LIN {X 0,Y 456.194,Z 627.483,A -85,B 0,C 180,E1 -8384.954,E2 -8384.954} C_VEL
LIN {X 0,Y 456.575,Z 617.149,A -85,B 0,C 180,E1 -8385.37,E2 -8385.37} C_VEL
LIN {X 0,Y 456.808,Z 606.428,A -85,B 0,C 180,E1 -8385.676,E2 -8385.676} C_VEL
LIN {X 0,Y 457.125,Z 587.235,A -85,B 0,C 180,E1 -8386.008,E2 -8386.008} C_VEL
LIN {X 0,Y 457.499,Z 519.528,A -85,B 0,C 180,E1 -8387.08,E2 -8387.08} C_VEL
LIN {X 0,Y 453.991,Z 499.289,A -85,B 0,C 180,E1 -8387.558,E2 -8387.558} C_VEL
LIN {X 0,Y 453.961,Z 498.233,A -85,B 0,C 180,E1 -8387.695,E2 -8387.695} C_VEL
LIN {X 0,Y 454.542,Z 486.824,A -85,B 0,C 180,E1 -8390.358,E2 -8390.358} C_VEL
LIN {X 0,Y 455.179,Z 474.408,A -85,B 0,C 180,E1 -8393.186,E2 -8393.186} C_VEL
LIN {X 0,Y 455.543,Z 466.02,A -85,B 0,C 180,E1 -8395.104,E2 -8395.104} C_VEL
LIN {X 0,Y 453.728,Z 455.779,A -85,B 0,C 180,E1 -8397.689,E2 -8397.689} C_VEL
LIN {X 0,Y 453.526,Z 454.578,A -85,B 0,C 180,E1 -8398.078,E2 -8398.078} C_VEL
LIN {X 0,Y 453.466,Z 454.501,A -85,B 0,C 180,E1 -8401.524,E2 -8401.524} C_VEL
LIN {X 0,Y 453.481,Z 454.495,A -85,B 0,C 180,E1 -8404.775,E2 -8404.775} C_VEL
LIN {X 0,Y 453.442,Z 454.504,A -85,B 0,C 180,E1 -8408.313,E2 -8408.313} C_VEL
LIN {X 0,Y 453.465,Z 454.484,A -85,B 0,C 180,E1 -8410.612,E2 -8410.612} C_VEL
LIN {X 0,Y 453.476,Z 454.496,A -85,B 0,C 180,E1 -8414.527,E2 -8414.527} C_VEL
LIN {X 0,Y 453.431,Z 454.507,A -85,B 0,C 180,E1 -8418.071,E2 -8418.071} C_VEL
LIN {X 0,Y 453.423,Z 454.498,A -85,B 0,C 180,E1 -8420.804,E2 -8420.804} C_VEL
LIN {X 0,Y 453.44,Z 454.505,A -85,B 0,C 180,E1 -8423.915,E2 -8423.915} C_VEL
LIN {X 0,Y 453.472,Z 454.489,A -85,B 0,C 180,E1 -8427.149,E2 -8427.149} C_VEL
LIN {X 0,Y 453.46,Z 454.5,A -85,B 0,C 180,E1 -8430.266,E2 -8430.266} C_VEL
LIN {X 0,Y 453.437,Z 454.486,A -85,B 0,C 180,E1 -8433.288,E2 -8433.288} C_VEL
LIN {X 0,Y 453.491,Z 454.497,A -85,B 0,C 180,E1 -8436.237,E2 -8436.237} C_VEL
LIN {X 0,Y 453.433,Z 454.495,A -85,B 0,C 180,E1 -8439.114,E2 -8439.114} C_VEL
LIN {X 0,Y 453.452,Z 454.485,A -85,B 0,C 180,E1 -8441.941,E2 -8441.941} C_VEL
LIN {X 0,Y 453.483,Z 454.492,A -85,B 0,C 180,E1 -8444.723,E2 -8444.723} C_VEL
LIN {X 0,Y 453.562,Z 454.482,A -85,B 0,C 180,E1 -8447.47,E2 -8447.47} C_VEL
LIN {X 0,Y 453.551,Z 454.467,A -85,B 0,C 180,E1 -8451.085,E2 -8451.085} C_VEL
LIN {X 0,Y 453.629,Z 454.474,A -85,B 0,C 180,E1 -8453.773,E2 -8453.773} C_VEL
LIN {X 0,Y 453.696,Z 454.465,A -85,B 0,C 180,E1 -8457.335,E2 -8457.335} C_VEL
LIN {X 0,Y 453.742,Z 454.449,A -85,B 0,C 180,E1 -8459.999,E2 -8459.999} C_VEL
LIN {X 0,Y 453.695,Z 454.464,A -85,B 0,C 180,E1 -8462.662,E2 -8462.662} C_VEL
LIN {X 0,Y 453.628,Z 454.479,A -85,B 0,C 180,E1 -8466.225,E2 -8466.225} C_VEL
LIN {X 0,Y 453.547,Z 454.473,A -85,B 0,C 180,E1 -8468.913,E2 -8468.913} C_VEL
LIN {X 0,Y 453.557,Z 454.484,A -85,B 0,C 180,E1 -8472.527,E2 -8472.527} C_VEL
LIN {X 0,Y 453.488,Z 454.495,A -85,B 0,C 180,E1 -8476.196,E2 -8476.196} C_VEL
LIN {X 0,Y 453.476,Z 454.478,A -85,B 0,C 180,E1 -8479.026,E2 -8479.026} C_VEL
LIN {X 0,Y 453.464,Z 454.495,A -85,B 0,C 180,E1 -8481.835,E2 -8481.835} C_VEL
LIN {X 0,Y 453.457,Z 454.495,A -85,B 0,C 180,E1 -8484.736,E2 -8484.736} C_VEL
LIN {X 0,Y 453.45,Z 454.49,A -85,B 0,C 180,E1 -8487.941,E2 -8487.941} C_VEL
LIN {X 0,Y 453.445,Z 454.499,A -85,B 0,C 180,E1 -8490.76,E2 -8490.76} C_VEL
LIN {X 0,Y 453.452,Z 454.495,A -85,B 0,C 180,E1 -8493.913,E2 -8493.913} C_VEL
LIN {X 0,Y 453.422,Z 454.501,A -85,B 0,C 180,E1 -8497.19,E2 -8497.19} C_VEL
LIN {X 0,Y 453.456,Z 454.491,A -85,B 0,C 180,E1 -8500.611,E2 -8500.611} C_VEL
LIN {X 0,Y 453.466,Z 454.495,A -85,B 0,C 180,E1 -8504.527,E2 -8504.527} C_VEL
LIN {X 0,Y 453.415,Z 454.481,A -85,B 0,C 180,E1 -8508.071,E2 -8508.071} C_VEL
LIN {X 0,Y 453.41,Z 454.502,A -85,B 0,C 180,E1 -8510.803,E2 -8510.803} C_VEL
LIN {X 0,Y 453.425,Z 454.497,A -85,B 0,C 180,E1 -8513.915,E2 -8513.915} C_VEL
LIN {X 0,Y 453.456,Z 454.495,A -85,B 0,C 180,E1 -8517.149,E2 -8517.149} C_VEL
LIN {X 0,Y 453.444,Z 454.491,A -85,B 0,C 180,E1 -8520.266,E2 -8520.266} C_VEL
LIN {X 0,Y 453.425,Z 454.503,A -85,B 0,C 180,E1 -8523.289,E2 -8523.289} C_VEL
LIN {X 0,Y 453.476,Z 454.501,A -85,B 0,C 180,E1 -8526.238,E2 -8526.238} C_VEL
LIN {X 0,Y 453.464,Z 454.498,A -85,B 0,C 180,E1 -8529.117,E2 -8529.117} C_VEL
LIN {X 0,Y 453.469,Z 454.502,A -85,B 0,C 180,E1 -8531.943,E2 -8531.943} C_VEL
LIN {X 0,Y 453.503,Z 454.495,A -85,B 0,C 180,E1 -8534.725,E2 -8534.725} C_VEL
LIN {X 0,Y 453.527,Z 454.494,A -85,B 0,C 180,E1 -8538.378,E2 -8538.378} C_VEL
LIN {X 0,Y 453.553,Z 454.488,A -85,B 0,C 180,E1 -8541.086,E2 -8541.086} C_VEL
LIN {X 0,Y 453.568,Z 454.487,A -85,B 0,C 180,E1 -8543.052,E2 -8543.052} C_VEL
LIN {X 0,Y 452.886,Z 454.575,A -85,B 0,C 180,E1 -8543.794,E2 -8543.794} C_VEL
LIN {X 0,Y 449.936,Z 454.939,A -85,B 0,C 180,E1 -8544.996,E2 -8544.996} C_VEL
LIN {X 0,Y 447.507,Z 455.245,A -85,B 0,C 180,E1 -8545.965,E2 -8545.965} C_VEL
LIN {X 0,Y 446.564,Z 455.361,A -85,B 0,C 180,E1 -8546.716,E2 -8546.716} C_VEL
LIN {X 0,Y 446.541,Z 455.362,A -85,B 0,C 180,E1 -8546.97,E2 -8546.97} C_VEL
LIN {X 0,Y 446.701,Z 455.345,A -85,B 0,C 180,E1 -8550,E2 -8550} C_VEL
LIN {X 0,Y 446.635,Z 455.351,A -85,B 0,C 180,E1 -8552.706,E2 -8552.706} C_VEL
LIN {X 0,Y 446.589,Z 455.359,A -85,B 0,C 180,E1 -8556.324,E2 -8556.324} C_VEL
LIN {X 0,Y 446.501,Z 455.367,A -85,B 0,C 180,E1 -8559.056,E2 -8559.056} C_VEL
LIN {X 0,Y 446.505,Z 455.367,A -85,B 0,C 180,E1 -8562.73,E2 -8562.73} C_VEL
LIN {X 0,Y 446.437,Z 455.378,A -85,B 0,C 180,E1 -8566.209,E2 -8566.209} C_VEL
LIN {X 0,Y 446.452,Z 455.373,A -85,B 0,C 180,E1 -8569.304,E2 -8569.304} C_VEL
LIN {X 0,Y 446.4,Z 455.382,A -85,B 0,C 180,E1 -8572.2,E2 -8572.2} C_VEL
LIN {X 0,Y 446.405,Z 455.378,A -85,B 0,C 180,E1 -8575.155,E2 -8575.155} C_VEL
LIN {X 0,Y 446.401,Z 455.373,A -85,B 0,C 180,E1 -8578.184,E2 -8578.184} C_VEL
LIN {X 0,Y 446.391,Z 455.378,A -85,B 0,C 180,E1 -8581.302,E2 -8581.302} C_VEL
LIN {X 0,Y 446.404,Z 455.361,A -85,B 0,C 180,E1 -8584.525,E2 -8584.525} C_VEL
LIN {X 0,Y 446.38,Z 455.385,A -85,B 0,C 180,E1 -8588.077,E2 -8588.077} C_VEL
LIN {X 0,Y 446.38,Z 455.36,A -85,B 0,C 180,E1 -8591.396,E2 -8591.396} C_VEL
LIN {X 0,Y 446.407,Z 455.372,A -85,B 0,C 180,E1 -8595.109,E2 -8595.109} C_VEL
LIN {X 0,Y 446.386,Z 455.371,A -85,B 0,C 180,E1 -8598.607,E2 -8598.607} C_VEL
LIN {X 0,Y 446.384,Z 455.385,A -85,B 0,C 180,E1 -8601.925,E2 -8601.925} C_VEL
LIN {X 0,Y 446.407,Z 455.368,A -85,B 0,C 180,E1 -8605.477,E2 -8605.477} C_VEL
LIN {X 0,Y 446.395,Z 455.377,A -85,B 0,C 180,E1 -8608.7,E2 -8608.7} C_VEL
LIN {X 0,Y 446.413,Z 455.368,A -85,B 0,C 180,E1 -8611.838,E2 -8611.838} C_VEL
LIN {X 0,Y 446.409,Z 455.372,A -85,B 0,C 180,E1 -8614.847,E2 -8614.847} C_VEL
LIN {X 0,Y 446.437,Z 455.369,A -85,B 0,C 180,E1 -8618.247,E2 -8618.247} C_VEL
LIN {X 0,Y 446.4,Z 455.363,A -85,B 0,C 180,E1 -8621.648,E2 -8621.648} C_VEL
LIN {X 0,Y 446.446,Z 455.372,A -85,B 0,C 180,E1 -8624.479,E2 -8624.479} C_VEL
LIN {X 0,Y 446.509,Z 455.361,A -85,B 0,C 180,E1 -8627.386,E2 -8627.386} C_VEL
LIN {X 0,Y 446.498,Z 455.351,A -85,B 0,C 180,E1 -8630.945,E2 -8630.945} C_VEL
LIN {X 0,Y 446.598,Z 455.353,A -85,B 0,C 180,E1 -8633.677,E2 -8633.677} C_VEL
LIN {X 0,Y 446.644,Z 455.342,A -85,B 0,C 180,E1 -8637.296,E2 -8637.296} C_VEL
LIN {X 0,Y 446.693,Z 455.326,A -85,B 0,C 180,E1 -8640.001,E2 -8640.001} C_VEL
LIN {X 0,Y 446.645,Z 455.343,A -85,B 0,C 180,E1 -8642.707,E2 -8642.707} C_VEL
LIN {X 0,Y 446.599,Z 455.348,A -85,B 0,C 180,E1 -8646.326,E2 -8646.326} C_VEL
LIN {X 0,Y 446.502,Z 455.345,A -85,B 0,C 180,E1 -8649.057,E2 -8649.057} C_VEL
LIN {X 0,Y 446.49,Z 455.362,A -85,B 0,C 180,E1 -8652.732,E2 -8652.732} C_VEL
LIN {X 0,Y 446.452,Z 455.364,A -85,B 0,C 180,E1 -8656.21,E2 -8656.21} C_VEL
LIN {X 0,Y 446.424,Z 455.358,A -85,B 0,C 180,E1 -8659.306,E2 -8659.306} C_VEL
LIN {X 0,Y 446.41,Z 455.378,A -85,B 0,C 180,E1 -8662.201,E2 -8662.201} C_VEL
LIN {X 0,Y 446.418,Z 455.368,A -85,B 0,C 180,E1 -8665.156,E2 -8665.156} C_VEL
LIN {X 0,Y 446.416,Z 455.374,A -85,B 0,C 180,E1 -8668.185,E2 -8668.185} C_VEL
LIN {X 0,Y 446.408,Z 455.376,A -85,B 0,C 180,E1 -8671.302,E2 -8671.302} C_VEL
LIN {X 0,Y 446.419,Z 455.369,A -85,B 0,C 180,E1 -8674.525,E2 -8674.525} C_VEL
LIN {X 0,Y 446.394,Z 455.379,A -85,B 0,C 180,E1 -8678.076,E2 -8678.076} C_VEL
LIN {X 0,Y 446.395,Z 455.377,A -85,B 0,C 180,E1 -8681.396,E2 -8681.396} C_VEL
LIN {X 0,Y 446.419,Z 455.372,A -85,B 0,C 180,E1 -8684.893,E2 -8684.893} C_VEL
LIN {X 0,Y 446.396,Z 455.364,A -85,B 0,C 180,E1 -8688.606,E2 -8688.606} C_VEL
LIN {X 0,Y 446.39,Z 455.38,A -85,B 0,C 180,E1 -8692.12,E2 -8692.12} C_VEL
LIN {X 0,Y 446.413,Z 455.377,A -85,B 0,C 180,E1 -8695.476,E2 -8695.476} C_VEL
LIN {X 0,Y 446.393,Z 455.381,A -85,B 0,C 180,E1 -8698.698,E2 -8698.698} C_VEL
LIN {X 0,Y 446.508,Z 455.533,A -85,B 0,C 180,E1 -8701.772,E2 -8701.772} C_VEL
LIN {X 0,Y 448.385,Z 465.875,A -85,B 0,C 180,E1 -8704.467,E2 -8704.467} C_VEL
LIN {X 0,Y 448.585,Z 469.327,A -85,B 0,C 180,E1 -8705.326,E2 -8705.326} C_VEL
LIN {X 0,Y 447.698,Z 484.427,A -85,B 0,C 180,E1 -8708.835,E2 -8708.835} C_VEL
LIN {X 0,Y 447.059,Z 496.641,A -85,B 0,C 180,E1 -8711.675,E2 -8711.675} C_VEL
LIN {X 0,Y 446.997,Z 498.636,A -85,B 0,C 180,E1 -8712.117,E2 -8712.117} C_VEL
LIN {X 0,Y 447.517,Z 502.122,A -85,B 0,C 180,E1 -8712.245,E2 -8712.245} C_VEL
LIN {X 0,Y 450.801,Z 520.895,A -85,B 0,C 180,E1 -8712.684,E2 -8712.684} C_VEL
LIN {X 0,Y 450.115,Z 603.591,A -85,B 0,C 180,E1 -8714.027,E2 -8714.027} C_VEL
LIN {X 0,Y 449.83,Z 613.508,A -85,B 0,C 180,E1 -8714.278,E2 -8714.278} C_VEL
LIN {X 0,Y 449.483,Z 623.498,A -85,B 0,C 180,E1 -8714.643,E2 -8714.643} C_VEL
LIN {X 0,Y 449.015,Z 633.857,A -85,B 0,C 180,E1 -8715.149,E2 -8715.149} C_VEL
LIN {X 0,Y 448.534,Z 643.004,A -85,B 0,C 180,E1 -8715.713,E2 -8715.713} C_VEL
LIN {X 0,Y 448.088,Z 652.01,A -85,B 0,C 180,E1 -8716.393,E2 -8716.393} C_VEL
LIN {X 0,Y 447.648,Z 660.495,A -85,B 0,C 180,E1 -8717.162,E2 -8717.162} C_VEL
LIN {X 0,Y 447.206,Z 668.165,A -85,B 0,C 180,E1 -8717.982,E2 -8717.982} C_VEL
LIN {X 0,Y 446.606,Z 676.962,A -85,B 0,C 180,E1 -8719.115,E2 -8719.115} C_VEL
LIN {X 0,Y 446.316,Z 682.955,A -85,B 0,C 180,E1 -8720.025,E2 -8720.025} C_VEL
LIN {X 0,Y 445.988,Z 689.266,A -85,B 0,C 180,E1 -8721.162,E2 -8721.162} C_VEL
LIN {X 0,Y 445.744,Z 694.54,A -85,B 0,C 180,E1 -8722.298,E2 -8722.298} C_VEL
LIN {X 0,Y 445.533,Z 699.632,A -85,B 0,C 180,E1 -8723.661,E2 -8723.661} C_VEL
LIN {X 0,Y 445.476,Z 703.595,A -85,B 0,C 180,E1 -8725.022,E2 -8725.022} C_VEL
LIN {X 0,Y 445.379,Z 706.524,A -85,B 0,C 180,E1 -8726.381,E2 -8726.381} C_VEL
LIN {X 0,Y 445.434,Z 708.024,A -85,B 0,C 180,E1 -8727.287,E2 -8727.287} C_VEL
LIN {X 0,Y 445.34,Z 709.541,A -85,B 0,C 180,E1 -8729.096,E2 -8729.096} C_VEL
LIN {X 0,Y 445.343,Z 709.82,A -85,B 0,C 180,E1 -8730,E2 -8730} C_VEL
LIN {X 0,Y 445.357,Z 708.948,A -85,B 0,C 180,E1 -8731.809,E2 -8731.809} C_VEL
LIN {X 0,Y 445.434,Z 708.024,A -85,B 0,C 180,E1 -8732.713,E2 -8732.713} C_VEL
LIN {X 0,Y 445.414,Z 704.681,A -85,B 0,C 180,E1 -8734.525,E2 -8734.525} C_VEL
LIN {X 0,Y 445.485,Z 702.471,A -85,B 0,C 180,E1 -8735.431,E2 -8735.431} C_VEL
LIN {X 0,Y 445.56,Z 698.291,A -85,B 0,C 180,E1 -8736.748,E2 -8736.748} C_VEL
LIN {X 0,Y 445.843,Z 692.544,A -85,B 0,C 180,E1 -8738.156,E2 -8738.156} C_VEL
LIN {X 0,Y 446.089,Z 686.89,A -85,B 0,C 180,E1 -8739.293,E2 -8739.293} C_VEL
LIN {X 0,Y 446.442,Z 680.084,A -85,B 0,C 180,E1 -8740.43,E2 -8740.43} C_VEL
LIN {X 0,Y 446.967,Z 671.867,A -85,B 0,C 180,E1 -8741.565,E2 -8741.565} C_VEL
LIN {X 0,Y 447.467,Z 664.038,A -85,B 0,C 180,E1 -8742.472,E2 -8742.472} C_VEL
LIN {X 0,Y 447.896,Z 655.918,A -85,B 0,C 180,E1 -8743.269,E2 -8743.269} C_VEL
LIN {X 0,Y 448.383,Z 646.186,A -85,B 0,C 180,E1 -8744.06,E2 -8744.06} C_VEL
LIN {X 0,Y 448.805,Z 637.793,A -85,B 0,C 180,E1 -8744.626,E2 -8744.626} C_VEL
LIN {X 0,Y 449.315,Z 627.286,A -85,B 0,C 180,E1 -8745.188,E2 -8745.188} C_VEL
LIN {X 0,Y 449.725,Z 616.953,A -85,B 0,C 180,E1 -8745.61,E2 -8745.61} C_VEL
LIN {X 0,Y 449.976,Z 606.232,A -85,B 0,C 180,E1 -8745.92,E2 -8745.92} C_VEL
LIN {X 0,Y 450.315,Z 587.039,A -85,B 0,C 180,E1 -8746.257,E2 -8746.257} C_VEL
LIN {X 0,Y 450.705,Z 520.339,A -85,B 0,C 180,E1 -8747.329,E2 -8747.329} C_VEL
LIN {X 0,Y 447.014,Z 499.093,A -85,B 0,C 180,E1 -8747.842,E2 -8747.842} C_VEL
LIN {X 0,Y 446.994,Z 497.666,A -85,B 0,C 180,E1 -8748.073,E2 -8748.073} C_VEL
LIN {X 0,Y 447.679,Z 485.631,A -85,B 0,C 180,E1 -8750.925,E2 -8750.925} C_VEL
LIN {X 0,Y 448.399,Z 472.173,A -85,B 0,C 180,E1 -8754.048,E2 -8754.048} C_VEL
LIN {X 0,Y 448.552,Z 466.927,A -85,B 0,C 180,E1 -8755.274,E2 -8755.274} C_VEL
LIN {X 0,Y 446.508,Z 455.53,A -85,B 0,C 180,E1 -8758.228,E2 -8758.228} C_VEL
LIN {X 0,Y 446.418,Z 455.381,A -85,B 0,C 180,E1 -8761.773,E2 -8761.773} C_VEL
LIN {X 0,Y 446.422,Z 455.377,A -85,B 0,C 180,E1 -8764.523,E2 -8764.523} C_VEL
LIN {X 0,Y 446.396,Z 455.383,A -85,B 0,C 180,E1 -8768.075,E2 -8768.075} C_VEL
LIN {X 0,Y 446.396,Z 455.364,A -85,B 0,C 180,E1 -8771.394,E2 -8771.394} C_VEL
LIN {X 0,Y 446.419,Z 455.372,A -85,B 0,C 180,E1 -8775.107,E2 -8775.107} C_VEL
LIN {X 0,Y 446.395,Z 455.377,A -85,B 0,C 180,E1 -8778.604,E2 -8778.604} C_VEL
LIN {X 0,Y 446.388,Z 455.382,A -85,B 0,C 180,E1 -8782.118,E2 -8782.118} C_VEL
LIN {X 0,Y 446.419,Z 455.369,A -85,B 0,C 180,E1 -8785.475,E2 -8785.475} C_VEL
LIN {X 0,Y 446.408,Z 455.376,A -85,B 0,C 180,E1 -8788.698,E2 -8788.698} C_VEL
LIN {X 0,Y 446.423,Z 455.372,A -85,B 0,C 180,E1 -8791.835,E2 -8791.835} C_VEL
LIN {X 0,Y 446.418,Z 455.368,A -85,B 0,C 180,E1 -8794.844,E2 -8794.844} C_VEL
LIN {X 0,Y 446.442,Z 455.372,A -85,B 0,C 180,E1 -8798.246,E2 -8798.246} C_VEL
LIN {X 0,Y 446.406,Z 455.361,A -85,B 0,C 180,E1 -8801.646,E2 -8801.646} C_VEL
LIN {X 0,Y 446.425,Z 455.373,A -85,B 0,C 180,E1 -8804.476,E2 -8804.476} C_VEL
LIN {X 0,Y 446.513,Z 455.36,A -85,B 0,C 180,E1 -8807.383,E2 -8807.383} C_VEL
LIN {X 0,Y 446.502,Z 455.345,A -85,B 0,C 180,E1 -8810.943,E2 -8810.943} C_VEL
LIN {X 0,Y 446.599,Z 455.348,A -85,B 0,C 180,E1 -8813.674,E2 -8813.674} C_VEL
LIN {X 0,Y 446.645,Z 455.343,A -85,B 0,C 180,E1 -8817.293,E2 -8817.293} C_VEL
LIN {X 0,Y 446.693,Z 455.326,A -85,B 0,C 180,E1 -8819.999,E2 -8819.999} C_VEL
LIN {X 0,Y 446.644,Z 455.342,A -85,B 0,C 180,E1 -8822.704,E2 -8822.704} C_VEL
LIN {X 0,Y 446.598,Z 455.353,A -85,B 0,C 180,E1 -8826.323,E2 -8826.323} C_VEL
LIN {X 0,Y 446.498,Z 455.351,A -85,B 0,C 180,E1 -8829.055,E2 -8829.055} C_VEL
LIN {X 0,Y 446.514,Z 455.359,A -85,B 0,C 180,E1 -8832.728,E2 -8832.728} C_VEL
LIN {X 0,Y 446.441,Z 455.372,A -85,B 0,C 180,E1 -8836.205,E2 -8836.205} C_VEL
LIN {X 0,Y 446.423,Z 455.357,A -85,B 0,C 180,E1 -8839.304,E2 -8839.304} C_VEL
LIN {X 0,Y 446.406,Z 455.38,A -85,B 0,C 180,E1 -8842.198,E2 -8842.198} C_VEL
LIN {X 0,Y 446.409,Z 455.372,A -85,B 0,C 180,E1 -8845.153,E2 -8845.153} C_VEL
LIN {X 0,Y 446.406,Z 455.369,A -85,B 0,C 180,E1 -8848.182,E2 -8848.182} C_VEL
LIN {X 0,Y 446.395,Z 455.377,A -85,B 0,C 180,E1 -8851.3,E2 -8851.3} C_VEL
LIN {X 0,Y 446.407,Z 455.368,A -85,B 0,C 180,E1 -8854.523,E2 -8854.523} C_VEL
LIN {X 0,Y 446.384,Z 455.385,A -85,B 0,C 180,E1 -8858.075,E2 -8858.075} C_VEL
LIN {X 0,Y 446.386,Z 455.371,A -85,B 0,C 180,E1 -8861.393,E2 -8861.393} C_VEL
LIN {X 0,Y 446.407,Z 455.372,A -85,B 0,C 180,E1 -8865.107,E2 -8865.107} C_VEL
LIN {X 0,Y 446.38,Z 455.36,A -85,B 0,C 180,E1 -8868.604,E2 -8868.604} C_VEL
LIN {X 0,Y 446.374,Z 455.386,A -85,B 0,C 180,E1 -8872.118,E2 -8872.118} C_VEL
LIN {X 0,Y 446.404,Z 455.361,A -85,B 0,C 180,E1 -8875.475,E2 -8875.475} C_VEL
LIN {X 0,Y 446.391,Z 455.378,A -85,B 0,C 180,E1 -8878.698,E2 -8878.698} C_VEL
LIN {X 0,Y 446.408,Z 455.373,A -85,B 0,C 180,E1 -8881.836,E2 -8881.836} C_VEL
LIN {X 0,Y 446.405,Z 455.378,A -85,B 0,C 180,E1 -8884.845,E2 -8884.845} C_VEL
LIN {X 0,Y 446.432,Z 455.378,A -85,B 0,C 180,E1 -8888.245,E2 -8888.245} C_VEL
LIN {X 0,Y 446.423,Z 455.379,A -85,B 0,C 180,E1 -8891.648,E2 -8891.648} C_VEL
LIN {X 0,Y 446.443,Z 455.376,A -85,B 0,C 180,E1 -8894.478,E2 -8894.478} C_VEL
LIN {X 0,Y 446.5,Z 455.368,A -85,B 0,C 180,E1 -8897.384,E2 -8897.384} C_VEL
LIN {X 0,Y 446.501,Z 455.367,A -85,B 0,C 180,E1 -8900.944,E2 -8900.944} C_VEL
LIN {X 0,Y 446.589,Z 455.359,A -85,B 0,C 180,E1 -8903.676,E2 -8903.676} C_VEL
LIN {X 0,Y 446.541,Z 455.362,A -85,B 0,C 180,E1 -8906.97,E2 -8906.97} C_VEL
LIN {X 0,Y 446.326,Z 455.39,A -85,B 0,C 180,E1 -8907.473,E2 -8907.473} C_VEL
LIN {X 0,Y 445.024,Z 455.554,A -85,B 0,C 180,E1 -8908.216,E2 -8908.216} C_VEL
LIN {X 0,Y 440.602,Z 456.106,A -85,B 0,C 180,E1 -8909.931,E2 -8909.931} C_VEL
LIN {X 0,Y 439.55,Z 456.235,A -85,B 0,C 180,E1 -8910.694,E2 -8910.694} C_VEL
LIN {X 0,Y 439.483,Z 456.242,A -85,B 0,C 180,E1 -8910.953,E2 -8910.953} C_VEL
LIN {X 0,Y 439.587,Z 456.229,A -85,B 0,C 180,E1 -8912.749,E2 -8912.749} C_VEL
LIN {X 0,Y 439.542,Z 456.236,A -85,B 0,C 180,E1 -8916.426,E2 -8916.426} C_VEL
LIN {X 0,Y 439.465,Z 456.244,A -85,B 0,C 180,E1 -8919.202,E2 -8919.202} C_VEL
LIN {X 0,Y 439.449,Z 456.245,A -85,B 0,C 180,E1 -8922.938,E2 -8922.938} C_VEL
LIN {X 0,Y 439.386,Z 456.255,A -85,B 0,C 180,E1 -8926.328,E2 -8926.328} C_VEL
LIN {X 0,Y 439.385,Z 456.256,A -85,B 0,C 180,E1 -8929.627,E2 -8929.627} C_VEL
LIN {X 0,Y 439.346,Z 456.259,A -85,B 0,C 180,E1 -8932.576,E2 -8932.576} C_VEL
LIN {X 0,Y 439.35,Z 456.259,A -85,B 0,C 180,E1 -8935.588,E2 -8935.588} C_VEL
LIN {X 0,Y 439.366,Z 456.245,A -85,B 0,C 180,E1 -8938.677,E2 -8938.677} C_VEL
LIN {X 0,Y 439.347,Z 456.26,A -85,B 0,C 180,E1 -8942.029,E2 -8942.029} C_VEL
LIN {X 0,Y 439.371,Z 456.237,A -85,B 0,C 180,E1 -8945.339,E2 -8945.339} C_VEL
LIN {X 0,Y 439.334,Z 456.257,A -85,B 0,C 180,E1 -8948.6,E2 -8948.6} C_VEL
LIN {X 0,Y 439.329,Z 456.234,A -85,B 0,C 180,E1 -8952.212,E2 -8952.212} C_VEL
LIN {X 0,Y 439.361,Z 456.25,A -85,B 0,C 180,E1 -8955.268,E2 -8955.268} C_VEL
LIN {X 0,Y 439.349,Z 456.247,A -85,B 0,C 180,E1 -8958.748,E2 -8958.748} C_VEL
LIN {X 0,Y 439.343,Z 456.258,A -85,B 0,C 180,E1 -8961.612,E2 -8961.612} C_VEL
LIN {X 0,Y 439.378,Z 456.242,A -85,B 0,C 180,E1 -8964.844,E2 -8964.844} C_VEL
LIN {X 0,Y 439.354,Z 456.26,A -85,B 0,C 180,E1 -8968.14,E2 -8968.14} C_VEL
LIN {X 0,Y 439.376,Z 456.247,A -85,B 0,C 180,E1 -8971.611,E2 -8971.611} C_VEL
LIN {X 0,Y 439.355,Z 456.253,A -85,B 0,C 180,E1 -8974.414,E2 -8974.414} C_VEL
LIN {X 0,Y 439.352,Z 456.255,A -85,B 0,C 180,E1 -8977.426,E2 -8977.426} C_VEL
LIN {X 0,Y 439.376,Z 456.234,A -85,B 0,C 180,E1 -8980.686,E2 -8980.686} C_VEL
LIN {X 0,Y 439.406,Z 456.251,A -85,B 0,C 180,E1 -8984.224,E2 -8984.224} C_VEL
LIN {X 0,Y 439.477,Z 456.236,A -85,B 0,C 180,E1 -8987.287,E2 -8987.287} C_VEL
LIN {X 0,Y 439.465,Z 456.227,A -85,B 0,C 180,E1 -8990.799,E2 -8990.799} C_VEL
LIN {X 0,Y 439.551,Z 456.229,A -85,B 0,C 180,E1 -8993.575,E2 -8993.575} C_VEL
LIN {X 0,Y 439.397,Z 456.25,A -85,B 0,C 180,E1 -8995.414,E2 -8995.414} C_VEL
LIN {X 0,Y 439.619,Z 456.208,A -85,B 0,C 180,E1 -8998.169,E2 -8998.169} C_VEL
LIN {X 0,Y 439.644,Z 456.203,A -85,B 0,C 180,E1 -9000.001,E2 -9000.001} C_VEL
LIN {X 0,Y 439.597,Z 456.221,A -85,B 0,C 180,E1 -9002.75,E2 -9002.75} C_VEL
LIN {X 0,Y 439.552,Z 456.225,A -85,B 0,C 180,E1 -9006.428,E2 -9006.428} C_VEL
LIN {X 0,Y 439.468,Z 456.221,A -85,B 0,C 180,E1 -9009.204,E2 -9009.204} C_VEL
LIN {X 0,Y 439.448,Z 456.239,A -85,B 0,C 180,E1 -9012.939,E2 -9012.939} C_VEL
LIN {X 0,Y 439.393,Z 456.241,A -85,B 0,C 180,E1 -9016.326,E2 -9016.326} C_VEL
LIN {X 0,Y 439.366,Z 456.24,A -85,B 0,C 180,E1 -9019.629,E2 -9019.629} C_VEL
LIN {X 0,Y 439.358,Z 456.253,A -85,B 0,C 180,E1 -9022.577,E2 -9022.577} C_VEL
LIN {X 0,Y 439.364,Z 456.248,A -85,B 0,C 180,E1 -9025.589,E2 -9025.589} C_VEL
LIN {X 0,Y 439.381,Z 456.248,A -85,B 0,C 180,E1 -9028.677,E2 -9028.677} C_VEL
LIN {X 0,Y 439.364,Z 456.252,A -85,B 0,C 180,E1 -9032.03,E2 -9032.03} C_VEL
LIN {X 0,Y 439.386,Z 456.245,A -85,B 0,C 180,E1 -9035.34,E2 -9035.34} C_VEL
LIN {X 0,Y 439.348,Z 456.251,A -85,B 0,C 180,E1 -9038.6,E2 -9038.6} C_VEL
LIN {X 0,Y 439.345,Z 456.258,A -85,B 0,C 180,E1 -9042.212,E2 -9042.212} C_VEL
LIN {X 0,Y 439.372,Z 456.251,A -85,B 0,C 180,E1 -9045.268,E2 -9045.268} C_VEL
LIN {X 0,Y 439.359,Z 456.24,A -85,B 0,C 180,E1 -9048.749,E2 -9048.749} C_VEL
LIN {X 0,Y 439.353,Z 456.258,A -85,B 0,C 180,E1 -9051.613,E2 -9051.613} C_VEL
LIN {X 0,Y 439.388,Z 456.25,A -85,B 0,C 180,E1 -9054.843,E2 -9054.843} C_VEL
LIN {X 0,Y 439.349,Z 456.259,A -85,B 0,C 180,E1 -9058.138,E2 -9058.138} C_VEL
LIN {X 0,Y 439.45,Z 456.457,A -85,B 0,C 180,E1 -9061.551,E2 -9061.551} C_VEL
LIN {X 0,Y 441.185,Z 465.728,A -85,B 0,C 180,E1 -9064.019,E2 -9064.019} C_VEL
LIN {X 0,Y 441.647,Z 469.934,A -85,B 0,C 180,E1 -9065.102,E2 -9065.102} C_VEL
LIN {X 0,Y 440.781,Z 484.254,A -85,B 0,C 180,E1 -9068.487,E2 -9068.487} C_VEL
LIN {X 0,Y 440.24,Z 494.5,A -85,B 0,C 180,E1 -9070.898,E2 -9070.898} C_VEL
LIN {X 0,Y 440.005,Z 498.44,A -85,B 0,C 180,E1 -9071.823,E2 -9071.823} C_VEL
LIN {X 0,Y 440.672,Z 502.437,A -85,B 0,C 180,E1 -9071.968,E2 -9071.968} C_VEL
LIN {X 0,Y 444.041,Z 522.403,A -85,B 0,C 180,E1 -9072.44,E2 -9072.44} C_VEL
LIN {X 0,Y 443.309,Z 603.395,A -85,B 0,C 180,E1 -9073.775,E2 -9073.775} C_VEL
LIN {X 0,Y 443.014,Z 613.313,A -85,B 0,C 180,E1 -9074.03,E2 -9074.03} C_VEL
LIN {X 0,Y 442.646,Z 623.302,A -85,B 0,C 180,E1 -9074.4,E2 -9074.4} C_VEL
LIN {X 0,Y 442.235,Z 631.691,A -85,B 0,C 180,E1 -9074.798,E2 -9074.798} C_VEL
LIN {X 0,Y 441.637,Z 642.807,A -85,B 0,C 180,E1 -9075.485,E2 -9075.485} C_VEL
LIN {X 0,Y 441.17,Z 651.813,A -85,B 0,C 180,E1 -9076.175,E2 -9076.175} C_VEL
LIN {X 0,Y 440.748,Z 659.713,A -85,B 0,C 180,E1 -9076.895,E2 -9076.895} C_VEL
LIN {X 0,Y 440.254,Z 667.969,A -85,B 0,C 180,E1 -9077.789,E2 -9077.789} C_VEL
LIN {X 0,Y 439.607,Z 676.765,A -85,B 0,C 180,E1 -9078.94,E2 -9078.94} C_VEL
LIN {X 0,Y 439.266,Z 682.757,A -85,B 0,C 180,E1 -9079.864,E2 -9079.864} C_VEL
LIN {X 0,Y 438.917,Z 689.069,A -85,B 0,C 180,E1 -9081.018,E2 -9081.018} C_VEL
LIN {X 0,Y 438.679,Z 694.343,A -85,B 0,C 180,E1 -9082.173,E2 -9082.173} C_VEL
LIN {X 0,Y 438.447,Z 699.663,A -85,B 0,C 180,E1 -9083.631,E2 -9083.631} C_VEL
LIN {X 0,Y 438.386,Z 703.398,A -85,B 0,C 180,E1 -9084.942,E2 -9084.942} C_VEL
LIN {X 0,Y 438.281,Z 706.328,A -85,B 0,C 180,E1 -9086.322,E2 -9086.322} C_VEL
LIN {X 0,Y 438.342,Z 707.828,A -85,B 0,C 180,E1 -9087.243,E2 -9087.243} C_VEL
LIN {X 0,Y 438.253,Z 709.345,A -85,B 0,C 180,E1 -9089.081,E2 -9089.081} C_VEL
LIN {X 0,Y 438.254,Z 709.624,A -85,B 0,C 180,E1 -9090,E2 -9090} C_VEL
LIN {X 0,Y 438.279,Z 708.752,A -85,B 0,C 180,E1 -9091.838,E2 -9091.838} C_VEL
LIN {X 0,Y 438.342,Z 707.828,A -85,B 0,C 180,E1 -9092.757,E2 -9092.757} C_VEL
LIN {X 0,Y 438.343,Z 704.485,A -85,B 0,C 180,E1 -9094.598,E2 -9094.598} C_VEL
LIN {X 0,Y 438.384,Z 702.274,A -85,B 0,C 180,E1 -9095.52,E2 -9095.52} C_VEL
LIN {X 0,Y 438.504,Z 697.921,A -85,B 0,C 180,E1 -9096.904,E2 -9096.904} C_VEL
LIN {X 0,Y 438.774,Z 692.347,A -85,B 0,C 180,E1 -9098.288,E2 -9098.288} C_VEL
LIN {X 0,Y 439.06,Z 686.693,A -85,B 0,C 180,E1 -9099.443,E2 -9099.443} C_VEL
LIN {X 0,Y 439.414,Z 679.887,A -85,B 0,C 180,E1 -9100.599,E2 -9100.599} C_VEL
LIN {X 0,Y 439.979,Z 671.669,A -85,B 0,C 180,E1 -9101.751,E2 -9101.751} C_VEL
LIN {X 0,Y 440.506,Z 663.841,A -85,B 0,C 180,E1 -9102.672,E2 -9102.672} C_VEL
LIN {X 0,Y 440.977,Z 655.016,A -85,B 0,C 180,E1 -9103.544,E2 -9103.544} C_VEL
LIN {X 0,Y 441.483,Z 645.989,A -85,B 0,C 180,E1 -9104.285,E2 -9104.285} C_VEL
LIN {X 0,Y 441.917,Z 637.596,A -85,B 0,C 180,E1 -9104.859,E2 -9104.859} C_VEL
LIN {X 0,Y 442.469,Z 627.09,A -85,B 0,C 180,E1 -9105.429,E2 -9105.429} C_VEL
LIN {X 0,Y 442.87,Z 616.756,A -85,B 0,C 180,E1 -9105.857,E2 -9105.857} C_VEL
LIN {X 0,Y 443.16,Z 606.036,A -85,B 0,C 180,E1 -9106.172,E2 -9106.172} C_VEL
LIN {X 0,Y 443.541,Z 585.054,A -85,B 0,C 180,E1 -9106.542,E2 -9106.542} C_VEL
LIN {X 0,Y 443.917,Z 521.182,A -85,B 0,C 180,E1 -9107.585,E2 -9107.585} C_VEL
LIN {X 0,Y 440.014,Z 498.828,A -85,B 0,C 180,E1 -9108.139,E2 -9108.139} C_VEL
LIN {X 0,Y 440.005,Z 498.063,A -85,B 0,C 180,E1 -9108.232,E2 -9108.232} C_VEL
LIN {X 0,Y 440.729,Z 485.464,A -85,B 0,C 180,E1 -9111.271,E2 -9111.271} C_VEL
LIN {X 0,Y 441.519,Z 472.033,A -85,B 0,C 180,E1 -9114.447,E2 -9114.447} C_VEL
LIN {X 0,Y 441.538,Z 467.834,A -85,B 0,C 180,E1 -9115.452,E2 -9115.452} C_VEL
LIN {X 0,Y 439.457,Z 456.479,A -85,B 0,C 180,E1 -9118.44,E2 -9118.44} C_VEL
LIN {X 0,Y 439.375,Z 456.252,A -85,B 0,C 180,E1 -9120.258,E2 -9120.258} C_VEL
LIN {X 0,Y 439.366,Z 456.253,A -85,B 0,C 180,E1 -9123.717,E2 -9123.717} C_VEL
LIN {X 0,Y 439.366,Z 456.248,A -85,B 0,C 180,E1 -9126.287,E2 -9126.287} C_VEL
LIN {X 0,Y 439.35,Z 456.256,A -85,B 0,C 180,E1 -9128.598,E2 -9128.598} C_VEL
LIN {X 0,Y 439.345,Z 456.251,A -85,B 0,C 180,E1 -9132.21,E2 -9132.21} C_VEL
LIN {X 0,Y 439.373,Z 456.25,A -85,B 0,C 180,E1 -9135.266,E2 -9135.266} C_VEL
LIN {X 0,Y 439.358,Z 456.252,A -85,B 0,C 180,E1 -9138.747,E2 -9138.747} C_VEL
LIN {X 0,Y 439.351,Z 456.252,A -85,B 0,C 180,E1 -9141.611,E2 -9141.611} C_VEL
LIN {X 0,Y 439.39,Z 456.244,A -85,B 0,C 180,E1 -9144.842,E2 -9144.842} C_VEL
LIN {X 0,Y 439.368,Z 456.254,A -85,B 0,C 180,E1 -9148.138,E2 -9148.138} C_VEL
LIN {X 0,Y 439.386,Z 456.249,A -85,B 0,C 180,E1 -9151.608,E2 -9151.608} C_VEL
LIN {X 0,Y 439.364,Z 456.248,A -85,B 0,C 180,E1 -9154.411,E2 -9154.411} C_VEL
LIN {X 0,Y 439.358,Z 456.253,A -85,B 0,C 180,E1 -9157.423,E2 -9157.423} C_VEL
LIN {X 0,Y 439.378,Z 456.236,A -85,B 0,C 180,E1 -9160.685,E2 -9160.685} C_VEL
LIN {X 0,Y 439.398,Z 456.249,A -85,B 0,C 180,E1 -9164.221,E2 -9164.221} C_VEL
LIN {X 0,Y 439.463,Z 456.238,A -85,B 0,C 180,E1 -9167.295,E2 -9167.295} C_VEL
LIN {X 0,Y 439.468,Z 456.221,A -85,B 0,C 180,E1 -9170.796,E2 -9170.796} C_VEL
LIN {X 0,Y 439.552,Z 456.225,A -85,B 0,C 180,E1 -9173.572,E2 -9173.572} C_VEL
LIN {X 0,Y 439.397,Z 456.249,A -85,B 0,C 180,E1 -9175.412,E2 -9175.412} C_VEL
LIN {X 0,Y 439.62,Z 456.216,A -85,B 0,C 180,E1 -9178.166,E2 -9178.166} C_VEL
LIN {X 0,Y 439.644,Z 456.203,A -85,B 0,C 180,E1 -9179.999,E2 -9179.999} C_VEL
LIN {X 0,Y 439.596,Z 456.219,A -85,B 0,C 180,E1 -9182.748,E2 -9182.748} C_VEL
LIN {X 0,Y 439.551,Z 456.229,A -85,B 0,C 180,E1 -9186.425,E2 -9186.425} C_VEL
LIN {X 0,Y 439.465,Z 456.227,A -85,B 0,C 180,E1 -9189.201,E2 -9189.201} C_VEL
LIN {X 0,Y 439.457,Z 456.238,A -85,B 0,C 180,E1 -9192.936,E2 -9192.936} C_VEL
LIN {X 0,Y 439.388,Z 456.249,A -85,B 0,C 180,E1 -9196.324,E2 -9196.324} C_VEL
LIN {X 0,Y 439.368,Z 456.236,A -85,B 0,C 180,E1 -9199.626,E2 -9199.626} C_VEL
LIN {X 0,Y 439.352,Z 456.255,A -85,B 0,C 180,E1 -9202.574,E2 -9202.574} C_VEL
LIN {X 0,Y 439.355,Z 456.253,A -85,B 0,C 180,E1 -9205.586,E2 -9205.586} C_VEL
LIN {X 0,Y 439.371,Z 456.248,A -85,B 0,C 180,E1 -9208.675,E2 -9208.675} C_VEL
LIN {X 0,Y 439.351,Z 456.259,A -85,B 0,C 180,E1 -9212.027,E2 -9212.027} C_VEL
LIN {X 0,Y 439.374,Z 456.243,A -85,B 0,C 180,E1 -9215.337,E2 -9215.337} C_VEL
LIN {X 0,Y 439.341,Z 456.256,A -85,B 0,C 180,E1 -9218.597,E2 -9218.597} C_VEL
LIN {X 0,Y 439.334,Z 456.26,A -85,B 0,C 180,E1 -9222.209,E2 -9222.209} C_VEL
LIN {X 0,Y 439.36,Z 456.25,A -85,B 0,C 180,E1 -9225.266,E2 -9225.266} C_VEL
LIN {X 0,Y 439.332,Z 456.241,A -85,B 0,C 180,E1 -9229.014,E2 -9229.014} C_VEL
LIN {X 0,Y 439.318,Z 456.259,A -85,B 0,C 180,E1 -9232.562,E2 -9232.562} C_VEL
LIN {X 0,Y 439.375,Z 456.236,A -85,B 0,C 180,E1 -9234.842,E2 -9234.842} C_VEL
LIN {X 0,Y 439.35,Z 456.261,A -85,B 0,C 180,E1 -9238.138,E2 -9238.138} C_VEL
LIN {X 0,Y 439.371,Z 456.246,A -85,B 0,C 180,E1 -9241.609,E2 -9241.609} C_VEL
LIN {X 0,Y 439.35,Z 456.259,A -85,B 0,C 180,E1 -9244.412,E2 -9244.412} C_VEL
LIN {X 0,Y 439.346,Z 456.259,A -85,B 0,C 180,E1 -9247.424,E2 -9247.424} C_VEL
LIN {X 0,Y 439.425,Z 456.249,A -85,B 0,C 180,E1 -9250.663,E2 -9250.663} C_VEL
LIN {X 0,Y 439.403,Z 456.254,A -85,B 0,C 180,E1 -9254.222,E2 -9254.222} C_VEL
LIN {X 0,Y 439.468,Z 456.243,A -85,B 0,C 180,E1 -9257.285,E2 -9257.285} C_VEL
LIN {X 0,Y 439.465,Z 456.244,A -85,B 0,C 180,E1 -9260.798,E2 -9260.798} C_VEL
LIN {X 0,Y 439.542,Z 456.236,A -85,B 0,C 180,E1 -9263.574,E2 -9263.574} C_VEL
LIN {X 0,Y 439.389,Z 456.255,A -85,B 0,C 180,E1 -9265.413,E2 -9265.413} C_VEL
LIN {X 0,Y 439.609,Z 456.228,A -85,B 0,C 180,E1 -9268.168,E2 -9268.168} C_VEL
LIN {X 0,Y 439.652,Z 456.223,A -85,B 0,C 180,E1 -9270,E2 -9270} C_VEL
LIN {X 0,Y 439.483,Z 456.242,A -85,B 0,C 180,E1 -9270.953,E2 -9270.953} C_VEL
LIN {X 0,Y 438.839,Z 456.324,A -85,B 0,C 180,E1 -9271.718,E2 -9271.718} C_VEL
LIN {X 0,Y 435.906,Z 456.688,A -85,B 0,C 180,E1 -9272.958,E2 -9272.958} C_VEL
LIN {X 0,Y 433.444,Z 456.997,A -85,B 0,C 180,E1 -9273.96,E2 -9273.96} C_VEL
LIN {X 0,Y 432.452,Z 457.119,A -85,B 0,C 180,E1 -9274.735,E2 -9274.735} C_VEL
LIN {X 0,Y 432.408,Z 457.123,A -85,B 0,C 180,E1 -9274.997,E2 -9274.997} C_VEL
LIN {X 0,Y 432.497,Z 457.113,A -85,B 0,C 180,E1 -9277.607,E2 -9277.607} C_VEL
LIN {X 0,Y 432.357,Z 457.13,A -85,B 0,C 180,E1 -9281.248,E2 -9281.248} C_VEL
LIN {X 0,Y 432.382,Z 457.126,A -85,B 0,C 180,E1 -9283.153,E2 -9283.153} C_VEL
LIN {X 0,Y 432.344,Z 457.132,A -85,B 0,C 180,E1 -9286.455,E2 -9286.455} C_VEL
LIN {X 0,Y 432.371,Z 457.129,A -85,B 0,C 180,E1 -9289.485,E2 -9289.485} C_VEL
LIN {X 0,Y 432.295,Z 457.136,A -85,B 0,C 180,E1 -9292.965,E2 -9292.965} C_VEL
LIN {X 0,Y 432.302,Z 457.139,A -85,B 0,C 180,E1 -9296.036,E2 -9296.036} C_VEL
LIN {X 0,Y 432.306,Z 457.121,A -85,B 0,C 180,E1 -9299.19,E2 -9299.19} C_VEL
LIN {X 0,Y 432.304,Z 457.132,A -85,B 0,C 180,E1 -9302.444,E2 -9302.444} C_VEL
LIN {X 0,Y 432.317,Z 457.12,A -85,B 0,C 180,E1 -9305.819,E2 -9305.819} C_VEL
LIN {X 0,Y 432.298,Z 457.133,A -85,B 0,C 180,E1 -9308.711,E2 -9308.711} C_VEL
LIN {X 0,Y 432.285,Z 457.11,A -85,B 0,C 180,E1 -9311.802,E2 -9311.802} C_VEL
LIN {X 0,Y 432.318,Z 457.126,A -85,B 0,C 180,E1 -9314.349,E2 -9314.349} C_VEL
LIN {X 0,Y 432.288,Z 457.134,A -85,B 0,C 180,E1 -9317.02,E2 -9317.02} C_VEL
LIN {X 0,Y 432.275,Z 457.131,A -85,B 0,C 180,E1 -9319.829,E2 -9319.829} C_VEL
LIN {X 0,Y 432.283,Z 457.135,A -85,B 0,C 180,E1 -9323.022,E2 -9323.022} C_VEL
LIN {X 0,Y 432.32,Z 457.125,A -85,B 0,C 180,E1 -9326.003,E2 -9326.003} C_VEL
LIN {X 0,Y 432.33,Z 457.132,A -85,B 0,C 180,E1 -9329.493,E2 -9329.493} C_VEL
LIN {X 0,Y 432.308,Z 457.123,A -85,B 0,C 180,E1 -9331.874,E2 -9331.874} C_VEL
LIN {X 0,Y 432.313,Z 457.128,A -85,B 0,C 180,E1 -9334.998,E2 -9334.998} C_VEL
LIN {X 0,Y 432.346,Z 457.126,A -85,B 0,C 180,E1 -9338.047,E2 -9338.047} C_VEL
LIN {X 0,Y 432.333,Z 457.11,A -85,B 0,C 180,E1 -9341.029,E2 -9341.029} C_VEL
LIN {X 0,Y 432.375,Z 457.126,A -85,B 0,C 180,E1 -9343.961,E2 -9343.961} C_VEL
LIN {X 0,Y 432.446,Z 457.11,A -85,B 0,C 180,E1 -9347.805,E2 -9347.805} C_VEL
LIN {X 0,Y 432.439,Z 457.105,A -85,B 0,C 180,E1 -9351.591,E2 -9351.591} C_VEL
LIN {X 0,Y 432.544,Z 457.104,A -85,B 0,C 180,E1 -9354.407,E2 -9354.407} C_VEL
LIN {X 0,Y 432.589,Z 457.083,A -85,B 0,C 180,E1 -9358.139,E2 -9358.139} C_VEL
LIN {X 0,Y 432.596,Z 457.08,A -85,B 0,C 180,E1 -9360.001,E2 -9360.001} C_VEL
LIN {X 0,Y 432.55,Z 457.099,A -85,B 0,C 180,E1 -9362.795,E2 -9362.795} C_VEL
LIN {X 0,Y 432.509,Z 457.101,A -85,B 0,C 180,E1 -9366.533,E2 -9366.533} C_VEL
LIN {X 0,Y 432.414,Z 457.099,A -85,B 0,C 180,E1 -9369.355,E2 -9369.355} C_VEL
LIN {X 0,Y 432.416,Z 457.115,A -85,B 0,C 180,E1 -9372.797,E2 -9372.797} C_VEL
LIN {X 0,Y 432.353,Z 457.117,A -85,B 0,C 180,E1 -9376.454,E2 -9376.454} C_VEL
LIN {X 0,Y 432.299,Z 457.124,A -85,B 0,C 180,E1 -9379.964,E2 -9379.964} C_VEL
LIN {X 0,Y 432.307,Z 457.13,A -85,B 0,C 180,E1 -9382.966,E2 -9382.966} C_VEL
LIN {X 0,Y 432.316,Z 457.119,A -85,B 0,C 180,E1 -9386.037,E2 -9386.037} C_VEL
LIN {X 0,Y 432.322,Z 457.128,A -85,B 0,C 180,E1 -9389.19,E2 -9389.19} C_VEL
LIN {X 0,Y 432.321,Z 457.125,A -85,B 0,C 180,E1 -9392.444,E2 -9392.444} C_VEL
LIN {X 0,Y 432.332,Z 457.129,A -85,B 0,C 180,E1 -9395.819,E2 -9395.819} C_VEL
LIN {X 0,Y 432.312,Z 457.127,A -85,B 0,C 180,E1 -9398.71,E2 -9398.71} C_VEL
LIN {X 0,Y 432.301,Z 457.137,A -85,B 0,C 180,E1 -9401.802,E2 -9401.802} C_VEL
LIN {X 0,Y 432.333,Z 457.129,A -85,B 0,C 180,E1 -9404.349,E2 -9404.349} C_VEL
LIN {X 0,Y 432.282,Z 457.135,A -85,B 0,C 180,E1 -9407.022,E2 -9407.022} C_VEL
LIN {X 0,Y 432.289,Z 457.124,A -85,B 0,C 180,E1 -9409.829,E2 -9409.829} C_VEL
LIN {X 0,Y 432.296,Z 457.131,A -85,B 0,C 180,E1 -9413.021,E2 -9413.021} C_VEL
LIN {X 0,Y 432.332,Z 457.132,A -85,B 0,C 180,E1 -9416.003,E2 -9416.003} C_VEL
LIN {X 0,Y 432.34,Z 457.129,A -85,B 0,C 180,E1 -9419.493,E2 -9419.493} C_VEL
LIN {X 0,Y 432.415,Z 457.309,A -85,B 0,C 180,E1 -9421.301,E2 -9421.301} C_VEL
LIN {X 0,Y 434.287,Z 467.536,A -85,B 0,C 180,E1 -9424.092,E2 -9424.092} C_VEL
LIN {X 0,Y 434.643,Z 471.65,A -85,B 0,C 180,E1 -9425.14,E2 -9425.14} C_VEL
LIN {X 0,Y 433.732,Z 486.149,A -85,B 0,C 180,E1 -9428.619,E2 -9428.619} C_VEL
LIN {X 0,Y 433.136,Z 496.249,A -85,B 0,C 180,E1 -9431.064,E2 -9431.064} C_VEL
LIN {X 0,Y 433.027,Z 498.245,A -85,B 0,C 180,E1 -9431.52,E2 -9431.52} C_VEL
LIN {X 0,Y 433.552,Z 501.421,A -85,B 0,C 180,E1 -9431.648,E2 -9431.648} C_VEL
LIN {X 0,Y 437.263,Z 523.103,A -85,B 0,C 180,E1 -9432.174,E2 -9432.174} C_VEL
LIN {X 0,Y 436.502,Z 603.199,A -85,B 0,C 180,E1 -9433.515,E2 -9433.515} C_VEL
LIN {X 0,Y 436.181,Z 613.116,A -85,B 0,C 180,E1 -9433.773,E2 -9433.773} C_VEL
LIN {X 0,Y 435.803,Z 623.105,A -85,B 0,C 180,E1 -9434.149,E2 -9434.149} C_VEL
LIN {X 0,Y 435.392,Z 631.495,A -85,B 0,C 180,E1 -9434.554,E2 -9434.554} C_VEL
LIN {X 0,Y 434.754,Z 642.611,A -85,B 0,C 180,E1 -9435.25,E2 -9435.25} C_VEL
LIN {X 0,Y 434.25,Z 651.616,A -85,B 0,C 180,E1 -9435.95,E2 -9435.95} C_VEL
LIN {X 0,Y 433.761,Z 659.952,A -85,B 0,C 180,E1 -9436.727,E2 -9436.727} C_VEL
LIN {X 0,Y 433.302,Z 667.772,A -85,B 0,C 180,E1 -9437.59,E2 -9437.59} C_VEL
LIN {X 0,Y 432.622,Z 676.568,A -85,B 0,C 180,E1 -9438.759,E2 -9438.759} C_VEL
LIN {X 0,Y 432.23,Z 682.559,A -85,B 0,C 180,E1 -9439.697,E2 -9439.697} C_VEL
LIN {X 0,Y 431.863,Z 688.871,A -85,B 0,C 180,E1 -9440.871,E2 -9440.871} C_VEL
LIN {X 0,Y 431.605,Z 694.146,A -85,B 0,C 180,E1 -9442.044,E2 -9442.044} C_VEL
LIN {X 0,Y 431.381,Z 699.238,A -85,B 0,C 180,E1 -9443.452,E2 -9443.452} C_VEL
LIN {X 0,Y 431.297,Z 703.201,A -85,B 0,C 180,E1 -9444.858,E2 -9444.858} C_VEL
LIN {X 0,Y 431.188,Z 706.131,A -85,B 0,C 180,E1 -9446.262,E2 -9446.262} C_VEL
LIN {X 0,Y 431.237,Z 707.631,A -85,B 0,C 180,E1 -9447.198,E2 -9447.198} C_VEL
LIN {X 0,Y 431.17,Z 709.149,A -85,B 0,C 180,E1 -9449.066,E2 -9449.066} C_VEL
LIN {X 0,Y 431.168,Z 709.428,A -85,B 0,C 180,E1 -9450,E2 -9450} C_VEL
LIN {X 0,Y 431.204,Z 708.556,A -85,B 0,C 180,E1 -9451.868,E2 -9451.868} C_VEL
LIN {X 0,Y 431.237,Z 707.631,A -85,B 0,C 180,E1 -9452.802,E2 -9452.802} C_VEL
LIN {X 0,Y 431.273,Z 704.289,A -85,B 0,C 180,E1 -9454.674,E2 -9454.674} C_VEL
LIN {X 0,Y 431.288,Z 700.966,A -85,B 0,C 180,E1 -9455.981,E2 -9455.981} C_VEL
LIN {X 0,Y 431.429,Z 697.724,A -85,B 0,C 180,E1 -9457.018,E2 -9457.018} C_VEL
LIN {X 0,Y 431.703,Z 692.149,A -85,B 0,C 180,E1 -9458.425,E2 -9458.425} C_VEL
LIN {X 0,Y 432.008,Z 686.495,A -85,B 0,C 180,E1 -9459.599,E2 -9459.599} C_VEL
LIN {X 0,Y 432.41,Z 679.69,A -85,B 0,C 180,E1 -9460.772,E2 -9460.772} C_VEL
LIN {X 0,Y 432.996,Z 671.472,A -85,B 0,C 180,E1 -9461.943,E2 -9461.943} C_VEL
LIN {X 0,Y 433.525,Z 663.644,A -85,B 0,C 180,E1 -9462.88,E2 -9462.88} C_VEL
LIN {X 0,Y 434.03,Z 654.97,A -85,B 0,C 180,E1 -9463.752,E2 -9463.752} C_VEL
LIN {X 0,Y 434.584,Z 645.792,A -85,B 0,C 180,E1 -9464.517,E2 -9464.517} C_VEL
LIN {X 0,Y 435.062,Z 637.4,A -85,B 0,C 180,E1 -9465.099,E2 -9465.099} C_VEL
LIN {X 0,Y 435.638,Z 626.894,A -85,B 0,C 180,E1 -9465.677,E2 -9465.677} C_VEL
LIN {X 0,Y 436.06,Z 616.56,A -85,B 0,C 180,E1 -9466.112,E2 -9466.112} C_VEL
LIN {X 0,Y 436.359,Z 605.84,A -85,B 0,C 180,E1 -9466.431,E2 -9466.431} C_VEL
LIN {X 0,Y 436.755,Z 584.858,A -85,B 0,C 180,E1 -9466.806,E2 -9466.806} C_VEL
LIN {X 0,Y 437.2,Z 522.24,A -85,B 0,C 180,E1 -9467.843,E2 -9467.843} C_VEL
LIN {X 0,Y 433.058,Z 498.595,A -85,B 0,C 180,E1 -9468.444,E2 -9468.444} C_VEL
LIN {X 0,Y 433.054,Z 497.299,A -85,B 0,C 180,E1 -9468.67,E2 -9468.67} C_VEL
LIN {X 0,Y 433.869,Z 484.269,A -85,B 0,C 180,E1 -9471.874,E2 -9471.874} C_VEL
LIN {X 0,Y 434.717,Z 470.772,A -85,B 0,C 180,E1 -9475.129,E2 -9475.129} C_VEL
LIN {X 0,Y 433.589,Z 463.552,A -85,B 0,C 180,E1 -9476.991,E2 -9476.991} C_VEL
LIN {X 0,Y 432.389,Z 457.239,A -85,B 0,C 180,E1 -9478.741,E2 -9478.741} C_VEL
LIN {X 0,Y 432.319,Z 457.135,A -85,B 0,C 180,E1 -9481.346,E2 -9481.346} C_VEL
LIN {X 0,Y 432.327,Z 457.131,A -85,B 0,C 180,E1 -9484.678,E2 -9484.678} C_VEL
LIN {X 0,Y 432.32,Z 457.137,A -85,B 0,C 180,E1 -9488.151,E2 -9488.151} C_VEL
LIN {X 0,Y 432.301,Z 457.122,A -85,B 0,C 180,E1 -9491.8,E2 -9491.8} C_VEL
LIN {X 0,Y 432.333,Z 457.131,A -85,B 0,C 180,E1 -9494.347,E2 -9494.347} C_VEL
LIN {X 0,Y 432.302,Z 457.132,A -85,B 0,C 180,E1 -9497.018,E2 -9497.018} C_VEL
LIN {X 0,Y 432.288,Z 457.133,A -85,B 0,C 180,E1 -9499.827,E2 -9499.827} C_VEL
LIN {X 0,Y 432.294,Z 457.133,A -85,B 0,C 180,E1 -9503.02,E2 -9503.02} C_VEL
LIN {X 0,Y 432.332,Z 457.122,A -85,B 0,C 180,E1 -9506.001,E2 -9506.001} C_VEL
LIN {X 0,Y 432.341,Z 457.128,A -85,B 0,C 180,E1 -9509.49,E2 -9509.49} C_VEL
LIN {X 0,Y 432.318,Z 457.127,A -85,B 0,C 180,E1 -9511.871,E2 -9511.871} C_VEL
LIN {X 0,Y 432.321,Z 457.123,A -85,B 0,C 180,E1 -9514.996,E2 -9514.996} C_VEL
LIN {X 0,Y 432.351,Z 457.13,A -85,B 0,C 180,E1 -9518.044,E2 -9518.044} C_VEL
LIN {X 0,Y 432.334,Z 457.111,A -85,B 0,C 180,E1 -9521.026,E2 -9521.026} C_VEL
LIN {X 0,Y 432.353,Z 457.121,A -85,B 0,C 180,E1 -9523.957,E2 -9523.957} C_VEL
LIN {X 0,Y 432.446,Z 457.116,A -85,B 0,C 180,E1 -9527.802,E2 -9527.802} C_VEL
LIN {X 0,Y 432.442,Z 457.097,A -85,B 0,C 180,E1 -9531.588,E2 -9531.588} C_VEL
LIN {X 0,Y 432.545,Z 457.105,A -85,B 0,C 180,E1 -9534.404,E2 -9534.404} C_VEL
LIN {X 0,Y 432.59,Z 457.091,A -85,B 0,C 180,E1 -9538.137,E2 -9538.137} C_VEL
LIN {X 0,Y 432.596,Z 457.08,A -85,B 0,C 180,E1 -9539.999,E2 -9539.999} C_VEL
LIN {X 0,Y 432.549,Z 457.097,A -85,B 0,C 180,E1 -9542.792,E2 -9542.792} C_VEL
LIN {X 0,Y 432.508,Z 457.106,A -85,B 0,C 180,E1 -9546.53,E2 -9546.53} C_VEL
LIN {X 0,Y 432.411,Z 457.105,A -85,B 0,C 180,E1 -9549.352,E2 -9549.352} C_VEL
LIN {X 0,Y 432.423,Z 457.114,A -85,B 0,C 180,E1 -9552.801,E2 -9552.801} C_VEL
LIN {X 0,Y 432.347,Z 457.124,A -85,B 0,C 180,E1 -9556.451,E2 -9556.451} C_VEL
LIN {X 0,Y 432.305,Z 457.118,A -85,B 0,C 180,E1 -9559.96,E2 -9559.96} C_VEL
LIN {X 0,Y 432.301,Z 457.132,A -85,B 0,C 180,E1 -9562.963,E2 -9562.963} C_VEL
LIN {X 0,Y 432.307,Z 457.127,A -85,B 0,C 180,E1 -9566.034,E2 -9566.034} C_VEL
LIN {X 0,Y 432.311,Z 457.126,A -85,B 0,C 180,E1 -9569.188,E2 -9569.188} C_VEL
LIN {X 0,Y 432.308,Z 457.131,A -85,B 0,C 180,E1 -9572.442,E2 -9572.442} C_VEL
LIN {X 0,Y 432.32,Z 457.125,A -85,B 0,C 180,E1 -9575.817,E2 -9575.817} C_VEL
LIN {X 0,Y 432.287,Z 457.134,A -85,B 0,C 180,E1 -9579.347,E2 -9579.347} C_VEL
LIN {X 0,Y 432.289,Z 457.13,A -85,B 0,C 180,E1 -9581.8,E2 -9581.8} C_VEL
LIN {X 0,Y 432.318,Z 457.13,A -85,B 0,C 180,E1 -9584.347,E2 -9584.347} C_VEL
LIN {X 0,Y 432.285,Z 457.115,A -85,B 0,C 180,E1 -9587.018,E2 -9587.018} C_VEL
LIN {X 0,Y 432.272,Z 457.125,A -85,B 0,C 180,E1 -9589.827,E2 -9589.827} C_VEL
LIN {X 0,Y 432.28,Z 457.135,A -85,B 0,C 180,E1 -9593.02,E2 -9593.02} C_VEL
LIN {X 0,Y 432.317,Z 457.117,A -85,B 0,C 180,E1 -9596.001,E2 -9596.001} C_VEL
LIN {X 0,Y 432.325,Z 457.131,A -85,B 0,C 180,E1 -9599.491,E2 -9599.491} C_VEL
LIN {X 0,Y 432.304,Z 457.129,A -85,B 0,C 180,E1 -9601.872,E2 -9601.872} C_VEL
LIN {X 0,Y 432.307,Z 457.134,A -85,B 0,C 180,E1 -9604.996,E2 -9604.996} C_VEL
LIN {X 0,Y 432.341,Z 457.134,A -85,B 0,C 180,E1 -9608.045,E2 -9608.045} C_VEL
LIN {X 0,Y 432.365,Z 457.128,A -85,B 0,C 180,E1 -9611.029,E2 -9611.029} C_VEL
LIN {X 0,Y 432.372,Z 457.13,A -85,B 0,C 180,E1 -9613.959,E2 -9613.959} C_VEL
LIN {X 0,Y 432.437,Z 457.121,A -85,B 0,C 180,E1 -9617.803,E2 -9617.803} C_VEL
LIN {X 0,Y 432.432,Z 457.122,A -85,B 0,C 180,E1 -9621.589,E2 -9621.589} C_VEL
LIN {X 0,Y 432.535,Z 457.109,A -85,B 0,C 180,E1 -9624.405,E2 -9624.405} C_VEL
LIN {X 0,Y 432.578,Z 457.104,A -85,B 0,C 180,E1 -9628.138,E2 -9628.138} C_VEL
LIN {X 0,Y 432.603,Z 457.101,A -85,B 0,C 180,E1 -9630,E2 -9630} C_VEL
LIN {X 0,Y 432.54,Z 457.107,A -85,B 0,C 180,E1 -9632.794,E2 -9632.794} C_VEL
LIN {X 0,Y 432.408,Z 457.123,A -85,B 0,C 180,E1 -9634.997,E2 -9634.997} C_VEL
LIN {X 0,Y 431.834,Z 457.197,A -85,B 0,C 180,E1 -9635.776,E2 -9635.776} C_VEL
LIN {X 0,Y 428.982,Z 457.551,A -85,B 0,C 180,E1 -9637.041,E2 -9637.041} C_VEL
LIN {X 0,Y 426.508,Z 457.86,A -85,B 0,C 180,E1 -9638.062,E2 -9638.062} C_VEL
LIN {X 0,Y 425.443,Z 457.991,A -85,B 0,C 180,E1 -9638.851,E2 -9638.851} C_VEL
LIN {X 0,Y 425.359,Z 458.001,A -85,B 0,C 180,E1 -9639.119,E2 -9639.119} C_VEL
LIN {X 0,Y 425.377,Z 457.999,A -85,B 0,C 180,E1 -9642.903,E2 -9642.903} C_VEL
LIN {X 0,Y 425.301,Z 458.009,A -85,B 0,C 180,E1 -9646.585,E2 -9646.585} C_VEL
LIN {X 0,Y 425.312,Z 458.009,A -85,B 0,C 180,E1 -9649.636,E2 -9649.636} C_VEL
LIN {X 0,Y 425.271,Z 458.014,A -85,B 0,C 180,E1 -9652.339,E2 -9652.339} C_VEL
LIN {X 0,Y 425.244,Z 458.016,A -85,B 0,C 180,E1 -9655.448,E2 -9655.448} C_VEL
LIN {X 0,Y 425.284,Z 457.997,A -85,B 0,C 180,E1 -9658.859,E2 -9658.859} C_VEL
LIN {X 0,Y 425.245,Z 458.018,A -85,B 0,C 180,E1 -9661.928,E2 -9661.928} C_VEL
LIN {X 0,Y 425.276,Z 457.992,A -85,B 0,C 180,E1 -9665.338,E2 -9665.338} C_VEL
LIN {X 0,Y 425.25,Z 458.01,A -85,B 0,C 180,E1 -9668.903,E2 -9668.903} C_VEL
LIN {X 0,Y 425.229,Z 457.987,A -85,B 0,C 180,E1 -9671.952,E2 -9671.952} C_VEL
LIN {X 0,Y 425.27,Z 458.005,A -85,B 0,C 180,E1 -9675.285,E2 -9675.285} C_VEL
LIN {X 0,Y 425.234,Z 458.005,A -85,B 0,C 180,E1 -9678.619,E2 -9678.619} C_VEL
LIN {X 0,Y 425.263,Z 458.008,A -85,B 0,C 180,E1 -9681.1,E2 -9681.1} C_VEL
LIN {X 0,Y 425.279,Z 457.998,A -85,B 0,C 180,E1 -9684.665,E2 -9684.665} C_VEL
LIN {X 0,Y 425.249,Z 458.017,A -85,B 0,C 180,E1 -9688.074,E2 -9688.074} C_VEL
LIN {X 0,Y 425.285,Z 458.002,A -85,B 0,C 180,E1 -9691.367,E2 -9691.367} C_VEL
LIN {X 0,Y 425.249,Z 458.01,A -85,B 0,C 180,E1 -9694.554,E2 -9694.554} C_VEL
LIN {X 0,Y 425.282,Z 458.011,A -85,B 0,C 180,E1 -9697.731,E2 -9697.731} C_VEL
LIN {X 0,Y 425.314,Z 457.984,A -85,B 0,C 180,E1 -9700.704,E2 -9700.704} C_VEL
LIN {X 0,Y 425.309,Z 458.002,A -85,B 0,C 180,E1 -9703.687,E2 -9703.687} C_VEL
LIN {X 0,Y 425.386,Z 457.991,A -85,B 0,C 180,E1 -9707.099,E2 -9707.099} C_VEL
LIN {X 0,Y 425.372,Z 457.982,A -85,B 0,C 180,E1 -9710.492,E2 -9710.492} C_VEL
LIN {X 0,Y 425.469,Z 457.982,A -85,B 0,C 180,E1 -9713.362,E2 -9713.362} C_VEL
LIN {X 0,Y 425.336,Z 458,A -85,B 0,C 180,E1 -9715.263,E2 -9715.263} C_VEL
LIN {X 0,Y 425.558,Z 457.959,A -85,B 0,C 180,E1 -9718.109,E2 -9718.109} C_VEL
LIN {X 0,Y 425.43,Z 457.976,A -85,B 0,C 180,E1 -9720.948,E2 -9720.948} C_VEL
LIN {X 0,Y 425.505,Z 457.976,A -85,B 0,C 180,E1 -9722.842,E2 -9722.842} C_VEL
LIN {X 0,Y 425.471,Z 457.977,A -85,B 0,C 180,E1 -9726.641,E2 -9726.641} C_VEL
LIN {X 0,Y 425.375,Z 457.976,A -85,B 0,C 180,E1 -9729.511,E2 -9729.511} C_VEL
LIN {X 0,Y 425.382,Z 457.991,A -85,B 0,C 180,E1 -9732.899,E2 -9732.899} C_VEL
LIN {X 0,Y 425.31,Z 457.993,A -85,B 0,C 180,E1 -9736.584,E2 -9736.584} C_VEL
LIN {X 0,Y 425.289,Z 457.992,A -85,B 0,C 180,E1 -9739.622,E2 -9739.622} C_VEL
LIN {X 0,Y 425.285,Z 458.008,A -85,B 0,C 180,E1 -9742.34,E2 -9742.34} C_VEL
LIN {X 0,Y 425.257,Z 458.005,A -85,B 0,C 180,E1 -9745.449,E2 -9745.449} C_VEL
LIN {X 0,Y 425.3,Z 458.002,A -85,B 0,C 180,E1 -9748.86,E2 -9748.86} C_VEL
LIN {X 0,Y 425.262,Z 458.01,A -85,B 0,C 180,E1 -9751.928,E2 -9751.928} C_VEL
LIN {X 0,Y 425.292,Z 458,A -85,B 0,C 180,E1 -9755.338,E2 -9755.338} C_VEL
LIN {X 0,Y 425.265,Z 458.005,A -85,B 0,C 180,E1 -9758.904,E2 -9758.904} C_VEL
LIN {X 0,Y 425.263,Z 458.016,A -85,B 0,C 180,E1 -9761.955,E2 -9761.955} C_VEL
LIN {X 0,Y 425.284,Z 458.006,A -85,B 0,C 180,E1 -9765.284,E2 -9765.284} C_VEL
LIN {X 0,Y 425.246,Z 457.997,A -85,B 0,C 180,E1 -9768.619,E2 -9768.619} C_VEL
LIN {X 0,Y 425.27,Z 458.009,A -85,B 0,C 180,E1 -9772.305,E2 -9772.305} C_VEL
LIN {X 0,Y 425.284,Z 458.013,A -85,B 0,C 180,E1 -9775.816,E2 -9775.816} C_VEL
LIN {X 0,Y 425.29,Z 458.008,A -85,B 0,C 180,E1 -9779.241,E2 -9779.241} C_VEL
LIN {X 0,Y 425.341,Z 458.203,A -85,B 0,C 180,E1 -9781.056,E2 -9781.056} C_VEL
LIN {X 0,Y 427.057,Z 467.391,A -85,B 0,C 180,E1 -9783.62,E2 -9783.62} C_VEL
LIN {X 0,Y 427.719,Z 472.51,A -85,B 0,C 180,E1 -9784.969,E2 -9784.969} C_VEL
LIN {X 0,Y 426.758,Z 487.01,A -85,B 0,C 180,E1 -9788.505,E2 -9788.505} C_VEL
LIN {X 0,Y 426.08,Z 498.05,A -85,B 0,C 180,E1 -9791.207,E2 -9791.207} C_VEL
LIN {X 0,Y 426.644,Z 501.503,A -85,B 0,C 180,E1 -9791.345,E2 -9791.345} C_VEL
LIN {X 0,Y 430.504,Z 523.71,A -85,B 0,C 180,E1 -9791.898,E2 -9791.898} C_VEL
LIN {X 0,Y 429.703,Z 603.003,A -85,B 0,C 180,E1 -9793.246,E2 -9793.246} C_VEL
LIN {X 0,Y 429.351,Z 612.919,A -85,B 0,C 180,E1 -9793.507,E2 -9793.507} C_VEL
LIN {X 0,Y 428.966,Z 622.909,A -85,B 0,C 180,E1 -9793.889,E2 -9793.889} C_VEL
LIN {X 0,Y 428.524,Z 631.298,A -85,B 0,C 180,E1 -9794.3,E2 -9794.3} C_VEL
LIN {X 0,Y 427.886,Z 642.414,A -85,B 0,C 180,E1 -9795.008,E2 -9795.008} C_VEL
LIN {X 0,Y 427.341,Z 651.419,A -85,B 0,C 180,E1 -9795.719,E2 -9795.719} C_VEL
LIN {X 0,Y 426.781,Z 660.162,A -85,B 0,C 180,E1 -9796.551,E2 -9796.551} C_VEL
LIN {X 0,Y 426.348,Z 667.575,A -85,B 0,C 180,E1 -9797.384,E2 -9797.384} C_VEL
LIN {X 0,Y 425.648,Z 676.371,A -85,B 0,C 180,E1 -9798.572,E2 -9798.572} C_VEL
LIN {X 0,Y 425.204,Z 682.362,A -85,B 0,C 180,E1 -9799.525,E2 -9799.525} C_VEL
LIN {X 0,Y 424.825,Z 688.674,A -85,B 0,C 180,E1 -9800.718,E2 -9800.718} C_VEL
LIN {X 0,Y 424.547,Z 693.949,A -85,B 0,C 180,E1 -9801.911,E2 -9801.911} C_VEL
LIN {X 0,Y 424.305,Z 699.041,A -85,B 0,C 180,E1 -9803.342,E2 -9803.342} C_VEL
LIN {X 0,Y 424.21,Z 703.005,A -85,B 0,C 180,E1 -9804.772,E2 -9804.772} C_VEL
LIN {X 0,Y 424.1,Z 705.935,A -85,B 0,C 180,E1 -9806.199,E2 -9806.199} C_VEL
LIN {X 0,Y 424.132,Z 707.435,A -85,B 0,C 180,E1 -9807.151,E2 -9807.151} C_VEL
LIN {X 0,Y 424.09,Z 708.954,A -85,B 0,C 180,E1 -9809.05,E2 -9809.05} C_VEL
LIN {X 0,Y 424.085,Z 709.232,A -85,B 0,C 180,E1 -9810,E2 -9810} C_VEL
LIN {X 0,Y 424.13,Z 708.361,A -85,B 0,C 180,E1 -9811.899,E2 -9811.899} C_VEL
LIN {X 0,Y 424.132,Z 707.435,A -85,B 0,C 180,E1 -9812.849,E2 -9812.849} C_VEL
LIN {X 0,Y 424.202,Z 704.093,A -85,B 0,C 180,E1 -9814.752,E2 -9814.752} C_VEL
LIN {X 0,Y 424.196,Z 701.88,A -85,B 0,C 180,E1 -9815.705,E2 -9815.705} C_VEL
LIN {X 0,Y 424.358,Z 697.527,A -85,B 0,C 180,E1 -9817.135,E2 -9817.135} C_VEL
LIN {X 0,Y 424.652,Z 691.952,A -85,B 0,C 180,E1 -9818.566,E2 -9818.566} C_VEL
LIN {X 0,Y 424.962,Z 686.298,A -85,B 0,C 180,E1 -9819.759,E2 -9819.759} C_VEL
LIN {X 0,Y 425.405,Z 679.493,A -85,B 0,C 180,E1 -9820.952,E2 -9820.952} C_VEL
LIN {X 0,Y 426.027,Z 671.275,A -85,B 0,C 180,E1 -9822.142,E2 -9822.142} C_VEL
LIN {X 0,Y 426.557,Z 663.446,A -85,B 0,C 180,E1 -9823.094,E2 -9823.094} C_VEL
LIN {X 0,Y 427.098,Z 655.213,A -85,B 0,C 180,E1 -9823.939,E2 -9823.939} C_VEL
LIN {X 0,Y 427.697,Z 645.595,A -85,B 0,C 180,E1 -9824.756,E2 -9824.756} C_VEL
LIN {X 0,Y 428.204,Z 637.204,A -85,B 0,C 180,E1 -9825.346,E2 -9825.346} C_VEL
LIN {X 0,Y 428.784,Z 626.697,A -85,B 0,C 180,E1 -9825.934,E2 -9825.934} C_VEL
LIN {X 0,Y 429.24,Z 616.364,A -85,B 0,C 180,E1 -9826.375,E2 -9826.375} C_VEL
LIN {X 0,Y 429.564,Z 605.644,A -85,B 0,C 180,E1 -9826.698,E2 -9826.698} C_VEL
LIN {X 0,Y 429.977,Z 584.662,A -85,B 0,C 180,E1 -9827.079,E2 -9827.079} C_VEL
LIN {X 0,Y 430.382,Z 522.755,A -85,B 0,C 180,E1 -9828.124,E2 -9828.124} C_VEL
LIN {X 0,Y 426.083,Z 498.324,A -85,B 0,C 180,E1 -9828.762,E2 -9828.762} C_VEL
LIN {X 0,Y 426.126,Z 497.009,A -85,B 0,C 180,E1 -9829.009,E2 -9829.009} C_VEL
LIN {X 0,Y 427.062,Z 482.846,A -85,B 0,C 180,E1 -9832.552,E2 -9832.552} C_VEL
LIN {X 0,Y 427.727,Z 471.506,A -85,B 0,C 180,E1 -9835.349,E2 -9835.349} C_VEL
LIN {X 0,Y 426.154,Z 462.395,A -85,B 0,C 180,E1 -9837.768,E2 -9837.768} C_VEL
LIN {X 0,Y 425.331,Z 458.105,A -85,B 0,C 180,E1 -9839.009,E2 -9839.009} C_VEL
LIN {X 0,Y 425.281,Z 458.004,A -85,B 0,C 180,E1 -9842.561,E2 -9842.561} C_VEL
LIN {X 0,Y 425.278,Z 458.003,A -85,B 0,C 180,E1 -9845.926,E2 -9845.926} C_VEL
LIN {X 0,Y 425.246,Z 458.011,A -85,B 0,C 180,E1 -9849.033,E2 -9849.033} C_VEL
LIN {X 0,Y 425.243,Z 458.002,A -85,B 0,C 180,E1 -9851.95,E2 -9851.95} C_VEL
LIN {X 0,Y 425.284,Z 458.005,A -85,B 0,C 180,E1 -9855.282,E2 -9855.282} C_VEL
LIN {X 0,Y 425.245,Z 458.011,A -85,B 0,C 180,E1 -9858.617,E2 -9858.617} C_VEL
LIN {X 0,Y 425.268,Z 458.014,A -85,B 0,C 180,E1 -9862.303,E2 -9862.303} C_VEL
LIN {X 0,Y 425.285,Z 457.999,A -85,B 0,C 180,E1 -9865.814,E2 -9865.814} C_VEL
LIN {X 0,Y 425.289,Z 458.006,A -85,B 0,C 180,E1 -9869.238,E2 -9869.238} C_VEL
LIN {X 0,Y 425.245,Z 457.999,A -85,B 0,C 180,E1 -9872.434,E2 -9872.434} C_VEL
LIN {X 0,Y 425.318,Z 457.998,A -85,B 0,C 180,E1 -9875.599,E2 -9875.599} C_VEL
LIN {X 0,Y 425.271,Z 458.004,A -85,B 0,C 180,E1 -9878.679,E2 -9878.679} C_VEL
LIN {X 0,Y 425.276,Z 457.99,A -85,B 0,C 180,E1 -9881.699,E2 -9881.699} C_VEL
LIN {X 0,Y 425.275,Z 458.006,A -85,B 0,C 180,E1 -9884.667,E2 -9884.667} C_VEL
LIN {X 0,Y 425.398,Z 457.991,A -85,B 0,C 180,E1 -9887.596,E2 -9887.596} C_VEL
LIN {X 0,Y 425.39,Z 457.974,A -85,B 0,C 180,E1 -9891.448,E2 -9891.448} C_VEL
LIN {X 0,Y 425.503,Z 457.983,A -85,B 0,C 180,E1 -9894.311,E2 -9894.311} C_VEL
LIN {X 0,Y 425.559,Z 457.967,A -85,B 0,C 180,E1 -9898.106,E2 -9898.106} C_VEL
LIN {X 0,Y 425.43,Z 457.97,A -85,B 0,C 180,E1 -9900.945,E2 -9900.945} C_VEL
LIN {X 0,Y 425.504,Z 457.974,A -85,B 0,C 180,E1 -9902.839,E2 -9902.839} C_VEL
LIN {X 0,Y 425.469,Z 457.982,A -85,B 0,C 180,E1 -9906.638,E2 -9906.638} C_VEL
LIN {X 0,Y 425.372,Z 457.982,A -85,B 0,C 180,E1 -9909.508,E2 -9909.508} C_VEL
LIN {X 0,Y 425.386,Z 457.991,A -85,B 0,C 180,E1 -9912.901,E2 -9912.901} C_VEL
LIN {X 0,Y 425.304,Z 458,A -85,B 0,C 180,E1 -9916.581,E2 -9916.581} C_VEL
LIN {X 0,Y 425.287,Z 457.989,A -85,B 0,C 180,E1 -9919.622,E2 -9919.622} C_VEL
LIN {X 0,Y 425.278,Z 458.011,A -85,B 0,C 180,E1 -9922.337,E2 -9922.337} C_VEL
LIN {X 0,Y 425.249,Z 458.01,A -85,B 0,C 180,E1 -9925.446,E2 -9925.446} C_VEL
LIN {X 0,Y 425.289,Z 458.001,A -85,B 0,C 180,E1 -9928.857,E2 -9928.857} C_VEL
LIN {X 0,Y 425.249,Z 458.017,A -85,B 0,C 180,E1 -9931.926,E2 -9931.926} C_VEL
LIN {X 0,Y 425.279,Z 457.998,A -85,B 0,C 180,E1 -9935.335,E2 -9935.335} C_VEL
LIN {X 0,Y 425.263,Z 458.008,A -85,B 0,C 180,E1 -9938.9,E2 -9938.9} C_VEL
LIN {X 0,Y 425.243,Z 458.013,A -85,B 0,C 180,E1 -9942.654,E2 -9942.654} C_VEL
LIN {X 0,Y 425.269,Z 458.005,A -85,B 0,C 180,E1 -9945.282,E2 -9945.282} C_VEL
LIN {X 0,Y 425.23,Z 457.99,A -85,B 0,C 180,E1 -9948.617,E2 -9948.617} C_VEL
LIN {X 0,Y 425.253,Z 458.014,A -85,B 0,C 180,E1 -9952.304,E2 -9952.304} C_VEL
LIN {X 0,Y 425.269,Z 457.993,A -85,B 0,C 180,E1 -9955.814,E2 -9955.814} C_VEL
LIN {X 0,Y 425.273,Z 458.008,A -85,B 0,C 180,E1 -9959.239,E2 -9959.239} C_VEL
LIN {X 0,Y 425.232,Z 458.018,A -85,B 0,C 180,E1 -9962.434,E2 -9962.434} C_VEL
LIN {X 0,Y 425.307,Z 458.009,A -85,B 0,C 180,E1 -9965.6,E2 -9965.6} C_VEL
LIN {X 0,Y 425.276,Z 458.011,A -85,B 0,C 180,E1 -9968.681,E2 -9968.681} C_VEL
LIN {X 0,Y 425.297,Z 458.011,A -85,B 0,C 180,E1 -9971.701,E2 -9971.701} C_VEL
LIN {X 0,Y 425.287,Z 458.01,A -85,B 0,C 180,E1 -9974.669,E2 -9974.669} C_VEL
LIN {X 0,Y 425.392,Z 457.999,A -85,B 0,C 180,E1 -9977.598,E2 -9977.598} C_VEL
LIN {X 0,Y 425.38,Z 458,A -85,B 0,C 180,E1 -9981.449,E2 -9981.449} C_VEL
LIN {X 0,Y 425.493,Z 457.987,A -85,B 0,C 180,E1 -9984.312,E2 -9984.312} C_VEL
LIN {X 0,Y 425.547,Z 457.98,A -85,B 0,C 180,E1 -9988.107,E2 -9988.107} C_VEL
LIN {X 0,Y 425.556,Z 457.979,A -85,B 0,C 180,E1 -9990,E2 -9990} C_VEL
LIN {X 0,Y 425.495,Z 457.985,A -85,B 0,C 180,E1 -9992.84,E2 -9992.84} C_VEL
LIN {X 0,Y 425.459,Z 457.99,A -85,B 0,C 180,E1 -9996.64,E2 -9996.64} C_VEL
LIN {X 0,Y 425.359,Z 458.001,A -85,B 0,C 180,E1 -9999.119,E2 -9999.119} C_VEL
LIN {X 0,Y 424.706,Z 458.085,A -85,B 0,C 180,E1 -9999.909,E2 -9999.909} C_VEL
LIN {X 0,Y 421.88,Z 458.436,A -85,B 0,C 180,E1 -10001.193,E2 -10001.193} C_VEL
LIN {X 0,Y 419.464,Z 458.737,A -85,B 0,C 180,E1 -10002.23,E2 -10002.23} C_VEL
LIN {X 0,Y 418.4,Z 458.868,A -85,B 0,C 180,E1 -10003.03,E2 -10003.03} C_VEL
LIN {X 0,Y 418.3,Z 458.881,A -85,B 0,C 180,E1 -10003.302,E2 -10003.302} C_VEL
LIN {X 0,Y 418.248,Z 458.888,A -85,B 0,C 180,E1 -10006.713,E2 -10006.713} C_VEL
LIN {X 0,Y 418.254,Z 458.888,A -85,B 0,C 180,E1 -10009.79,E2 -10009.79} C_VEL
LIN {X 0,Y 418.212,Z 458.891,A -85,B 0,C 180,E1 -10012.737,E2 -10012.737} C_VEL
LIN {X 0,Y 418.209,Z 458.894,A -85,B 0,C 180,E1 -10015.908,E2 -10015.908} C_VEL
LIN {X 0,Y 418.241,Z 458.872,A -85,B 0,C 180,E1 -10019.163,E2 -10019.163} C_VEL
LIN {X 0,Y 418.235,Z 458.882,A -85,B 0,C 180,E1 -10022.843,E2 -10022.843} C_VEL
LIN {X 0,Y 418.223,Z 458.882,A -85,B 0,C 180,E1 -10026.237,E2 -10026.237} C_VEL
LIN {X 0,Y 418.178,Z 458.887,A -85,B 0,C 180,E1 -10029.69,E2 -10029.69} C_VEL
LIN {X 0,Y 418.194,Z 458.863,A -85,B 0,C 180,E1 -10032.319,E2 -10032.319} C_VEL
LIN {X 0,Y 418.22,Z 458.883,A -85,B 0,C 180,E1 -10035.109,E2 -10035.109} C_VEL
LIN {X 0,Y 418.205,Z 458.891,A -85,B 0,C 180,E1 -10037.765,E2 -10037.765} C_VEL
LIN {X 0,Y 418.221,Z 458.888,A -85,B 0,C 180,E1 -10041.557,E2 -10041.557} C_VEL
LIN {X 0,Y 418.237,Z 458.875,A -85,B 0,C 180,E1 -10045.159,E2 -10045.159} C_VEL
LIN {X 0,Y 418.23,Z 458.884,A -85,B 0,C 180,E1 -10047.473,E2 -10047.473} C_VEL
LIN {X 0,Y 418.248,Z 458.877,A -85,B 0,C 180,E1 -10050.899,E2 -10050.899} C_VEL
LIN {X 0,Y 418.207,Z 458.884,A -85,B 0,C 180,E1 -10054.094,E2 -10054.094} C_VEL
LIN {X 0,Y 418.218,Z 458.887,A -85,B 0,C 180,E1 -10057.265,E2 -10057.265} C_VEL
LIN {X 0,Y 418.241,Z 458.866,A -85,B 0,C 180,E1 -10060.364,E2 -10060.364} C_VEL
LIN {X 0,Y 418.271,Z 458.876,A -85,B 0,C 180,E1 -10063.405,E2 -10063.405} C_VEL
LIN {X 0,Y 418.338,Z 458.868,A -85,B 0,C 180,E1 -10067.002,E2 -10067.002} C_VEL
LIN {X 0,Y 418.312,Z 458.859,A -85,B 0,C 180,E1 -10070.33,E2 -10070.33} C_VEL
LIN {X 0,Y 418.434,Z 458.857,A -85,B 0,C 180,E1 -10073.25,E2 -10073.25} C_VEL
LIN {X 0,Y 418.306,Z 458.876,A -85,B 0,C 180,E1 -10075.183,E2 -10075.183} C_VEL
LIN {X 0,Y 418.527,Z 458.835,A -85,B 0,C 180,E1 -10078.077,E2 -10078.077} C_VEL
LIN {X 0,Y 418.4,Z 458.851,A -85,B 0,C 180,E1 -10080.964,E2 -10080.964} C_VEL
LIN {X 0,Y 418.462,Z 458.854,A -85,B 0,C 180,E1 -10082.889,E2 -10082.889} C_VEL
LIN {X 0,Y 418.464,Z 458.86,A -85,B 0,C 180,E1 -10085.785,E2 -10085.785} C_VEL
LIN {X 0,Y 418.362,Z 458.848,A -85,B 0,C 180,E1 -10088.697,E2 -10088.697} C_VEL
LIN {X 0,Y 418.296,Z 458.869,A -85,B 0,C 180,E1 -10091.633,E2 -10091.633} C_VEL
LIN {X 0,Y 418.274,Z 458.88,A -85,B 0,C 180,E1 -10093.607,E2 -10093.607} C_VEL
LIN {X 0,Y 418.249,Z 458.872,A -85,B 0,C 180,E1 -10096.708,E2 -10096.708} C_VEL
LIN {X 0,Y 418.233,Z 458.872,A -85,B 0,C 180,E1 -10099.777,E2 -10099.777} C_VEL
LIN {X 0,Y 418.225,Z 458.885,A -85,B 0,C 180,E1 -10102.738,E2 -10102.738} C_VEL
LIN {X 0,Y 418.217,Z 458.875,A -85,B 0,C 180,E1 -10105.909,E2 -10105.909} C_VEL
LIN {X 0,Y 418.256,Z 458.879,A -85,B 0,C 180,E1 -10109.164,E2 -10109.164} C_VEL
LIN {X 0,Y 418.251,Z 458.875,A -85,B 0,C 180,E1 -10112.843,E2 -10112.843} C_VEL
LIN {X 0,Y 418.239,Z 458.888,A -85,B 0,C 180,E1 -10116.238,E2 -10116.238} C_VEL
LIN {X 0,Y 418.193,Z 458.887,A -85,B 0,C 180,E1 -10119.69,E2 -10119.69} C_VEL
LIN {X 0,Y 418.206,Z 458.89,A -85,B 0,C 180,E1 -10122.318,E2 -10122.318} C_VEL
LIN {X 0,Y 418.235,Z 458.884,A -85,B 0,C 180,E1 -10125.109,E2 -10125.109} C_VEL
LIN {X 0,Y 418.209,Z 458.883,A -85,B 0,C 180,E1 -10127.764,E2 -10127.764} C_VEL
LIN {X 0,Y 418.198,Z 458.889,A -85,B 0,C 180,E1 -10130.63,E2 -10130.63} C_VEL
LIN {X 0,Y 418.237,Z 458.878,A -85,B 0,C 180,E1 -10133.976,E2 -10133.976} C_VEL
LIN {X 0,Y 418.243,Z 458.88,A -85,B 0,C 180,E1 -10137.161,E2 -10137.161} C_VEL
LIN {X 0,Y 418.268,Z 459.018,A -85,B 0,C 180,E1 -10140.77,E2 -10140.77} C_VEL
LIN {X 0,Y 420.194,Z 469.197,A -85,B 0,C 180,E1 -10143.69,E2 -10143.69} C_VEL
LIN {X 0,Y 420.763,Z 473.746,A -85,B 0,C 180,E1 -10144.887,E2 -10144.887} C_VEL
LIN {X 0,Y 419.785,Z 487.871,A -85,B 0,C 180,E1 -10148.388,E2 -10148.388} C_VEL
LIN {X 0,Y 419.112,Z 497.851,A -85,B 0,C 180,E1 -10150.883,E2 -10150.883} C_VEL
LIN {X 0,Y 419.661,Z 501.207,A -85,B 0,C 180,E1 -10151.021,E2 -10151.021} C_VEL
LIN {X 0,Y 423.705,Z 524.098,A -85,B 0,C 180,E1 -10151.608,E2 -10151.608} C_VEL
LIN {X 0,Y 422.906,Z 602.806,A -85,B 0,C 180,E1 -10152.969,E2 -10152.969} C_VEL
LIN {X 0,Y 422.562,Z 612.724,A -85,B 0,C 180,E1 -10153.234,E2 -10153.234} C_VEL
LIN {X 0,Y 422.148,Z 622.713,A -85,B 0,C 180,E1 -10153.622,E2 -10153.622} C_VEL
LIN {X 0,Y 421.57,Z 633.07,A -85,B 0,C 180,E1 -10154.158,E2 -10154.158} C_VEL
LIN {X 0,Y 421.005,Z 642.217,A -85,B 0,C 180,E1 -10154.757,E2 -10154.757} C_VEL
LIN {X 0,Y 420.438,Z 651.222,A -85,B 0,C 180,E1 -10155.479,E2 -10155.479} C_VEL
LIN {X 0,Y 419.884,Z 659.609,A -85,B 0,C 180,E1 -10156.286,E2 -10156.286} C_VEL
LIN {X 0,Y 419.393,Z 667.378,A -85,B 0,C 180,E1 -10157.171,E2 -10157.171} C_VEL
LIN {X 0,Y 418.654,Z 676.174,A -85,B 0,C 180,E1 -10158.379,E2 -10158.379} C_VEL
LIN {X 0,Y 418.179,Z 682.164,A -85,B 0,C 180,E1 -10159.347,E2 -10159.347} C_VEL
LIN {X 0,Y 417.788,Z 688.477,A -85,B 0,C 180,E1 -10160.56,E2 -10160.56} C_VEL
LIN {X 0,Y 417.482,Z 693.751,A -85,B 0,C 180,E1 -10161.773,E2 -10161.773} C_VEL
LIN {X 0,Y 417.239,Z 698.845,A -85,B 0,C 180,E1 -10163.229,E2 -10163.229} C_VEL
LIN {X 0,Y 417.125,Z 702.808,A -85,B 0,C 180,E1 -10164.683,E2 -10164.683} C_VEL
LIN {X 0,Y 417.015,Z 705.739,A -85,B 0,C 180,E1 -10166.135,E2 -10166.135} C_VEL
LIN {X 0,Y 417.029,Z 707.238,A -85,B 0,C 180,E1 -10167.102,E2 -10167.102} C_VEL
LIN {X 0,Y 417.012,Z 708.758,A -85,B 0,C 180,E1 -10169.034,E2 -10169.034} C_VEL
LIN {X 0,Y 417.005,Z 709.036,A -85,B 0,C 180,E1 -10170,E2 -10170} C_VEL
LIN {X 0,Y 417.058,Z 708.165,A -85,B 0,C 180,E1 -10171.931,E2 -10171.931} C_VEL
LIN {X 0,Y 417.029,Z 707.238,A -85,B 0,C 180,E1 -10172.898,E2 -10172.898} C_VEL
LIN {X 0,Y 417.11,Z 703.896,A -85,B 0,C 180,E1 -10174.833,E2 -10174.833} C_VEL
LIN {X 0,Y 417.145,Z 700.348,A -85,B 0,C 180,E1 -10176.261,E2 -10176.261} C_VEL
LIN {X 0,Y 417.381,Z 695.541,A -85,B 0,C 180,E1 -10177.742,E2 -10177.742} C_VEL
LIN {X 0,Y 417.702,Z 689.569,A -85,B 0,C 180,E1 -10179.198,E2 -10179.198} C_VEL
LIN {X 0,Y 418.115,Z 683.477,A -85,B 0,C 180,E1 -10180.41,E2 -10180.41} C_VEL
LIN {X 0,Y 418.515,Z 677.734,A -85,B 0,C 180,E1 -10181.38,E2 -10181.38} C_VEL
LIN {X 0,Y 419.062,Z 671.078,A -85,B 0,C 180,E1 -10182.347,E2 -10182.347} C_VEL
LIN {X 0,Y 419.619,Z 663.249,A -85,B 0,C 180,E1 -10183.314,E2 -10183.314} C_VEL
LIN {X 0,Y 420.217,Z 654.422,A -85,B 0,C 180,E1 -10184.228,E2 -10184.228} C_VEL
LIN {X 0,Y 420.819,Z 645.399,A -85,B 0,C 180,E1 -10185.002,E2 -10185.002} C_VEL
LIN {X 0,Y 421.368,Z 637.008,A -85,B 0,C 180,E1 -10185.602,E2 -10185.602} C_VEL
LIN {X 0,Y 421.961,Z 626.501,A -85,B 0,C 180,E1 -10186.199,E2 -10186.199} C_VEL
LIN {X 0,Y 422.441,Z 616.168,A -85,B 0,C 180,E1 -10186.646,E2 -10186.646} C_VEL
LIN {X 0,Y 422.784,Z 605.448,A -85,B 0,C 180,E1 -10186.974,E2 -10186.974} C_VEL
LIN {X 0,Y 423.201,Z 584.466,A -85,B 0,C 180,E1 -10187.361,E2 -10187.361} C_VEL
LIN {X 0,Y 423.662,Z 523.783,A -85,B 0,C 180,E1 -10188.4,E2 -10188.4} C_VEL
LIN {X 0,Y 419.132,Z 498.127,A -85,B 0,C 180,E1 -10189.085,E2 -10189.085} C_VEL
LIN {X 0,Y 419.155,Z 496.811,A -85,B 0,C 180,E1 -10189.338,E2 -10189.338} C_VEL
LIN {X 0,Y 420.072,Z 483.935,A -85,B 0,C 180,E1 -10192.631,E2 -10192.631} C_VEL
LIN {X 0,Y 420.777,Z 473.984,A -85,B 0,C 180,E1 -10195.118,E2 -10195.118} C_VEL
LIN {X 0,Y 420.269,Z 469.486,A -85,B 0,C 180,E1 -10196.305,E2 -10196.305} C_VEL
LIN {X 0,Y 418.289,Z 459.043,A -85,B 0,C 180,E1 -10199.211,E2 -10199.211} C_VEL
LIN {X 0,Y 418.254,Z 458.879,A -85,B 0,C 180,E1 -10202.842,E2 -10202.842} C_VEL
LIN {X 0,Y 418.241,Z 458.878,A -85,B 0,C 180,E1 -10206.236,E2 -10206.236} C_VEL
LIN {X 0,Y 418.195,Z 458.885,A -85,B 0,C 180,E1 -10209.688,E2 -10209.688} C_VEL
LIN {X 0,Y 418.21,Z 458.884,A -85,B 0,C 180,E1 -10212.317,E2 -10212.317} C_VEL
LIN {X 0,Y 418.235,Z 458.883,A -85,B 0,C 180,E1 -10215.107,E2 -10215.107} C_VEL
LIN {X 0,Y 418.218,Z 458.89,A -85,B 0,C 180,E1 -10217.763,E2 -10217.763} C_VEL
LIN {X 0,Y 418.227,Z 458.883,A -85,B 0,C 180,E1 -10221.554,E2 -10221.554} C_VEL
LIN {X 0,Y 418.249,Z 458.876,A -85,B 0,C 180,E1 -10225.157,E2 -10225.157} C_VEL
LIN {X 0,Y 418.243,Z 458.877,A -85,B 0,C 180,E1 -10227.47,E2 -10227.47} C_VEL
LIN {X 0,Y 418.259,Z 458.879,A -85,B 0,C 180,E1 -10230.897,E2 -10230.897} C_VEL
LIN {X 0,Y 418.217,Z 458.875,A -85,B 0,C 180,E1 -10234.091,E2 -10234.091} C_VEL
LIN {X 0,Y 418.225,Z 458.885,A -85,B 0,C 180,E1 -10237.262,E2 -10237.262} C_VEL
LIN {X 0,Y 418.243,Z 458.869,A -85,B 0,C 180,E1 -10240.361,E2 -10240.361} C_VEL
LIN {X 0,Y 418.277,Z 458.869,A -85,B 0,C 180,E1 -10243.402,E2 -10243.402} C_VEL
LIN {X 0,Y 418.343,Z 458.869,A -85,B 0,C 180,E1 -10247.384,E2 -10247.384} C_VEL
LIN {X 0,Y 418.315,Z 458.855,A -85,B 0,C 180,E1 -10250.327,E2 -10250.327} C_VEL
LIN {X 0,Y 418.436,Z 458.853,A -85,B 0,C 180,E1 -10253.247,E2 -10253.247} C_VEL
LIN {X 0,Y 418.307,Z 458.875,A -85,B 0,C 180,E1 -10255.18,E2 -10255.18} C_VEL
LIN {X 0,Y 418.528,Z 458.843,A -85,B 0,C 180,E1 -10258.074,E2 -10258.074} C_VEL
LIN {X 0,Y 418.4,Z 458.845,A -85,B 0,C 180,E1 -10260.961,E2 -10260.961} C_VEL
LIN {X 0,Y 418.461,Z 458.851,A -85,B 0,C 180,E1 -10262.887,E2 -10262.887} C_VEL
LIN {X 0,Y 418.43,Z 458.858,A -85,B 0,C 180,E1 -10266.532,E2 -10266.532} C_VEL
LIN {X 0,Y 418.359,Z 458.855,A -85,B 0,C 180,E1 -10268.694,E2 -10268.694} C_VEL
LIN {X 0,Y 418.346,Z 458.869,A -85,B 0,C 180,E1 -10272.613,E2 -10272.613} C_VEL
LIN {X 0,Y 418.239,Z 458.886,A -85,B 0,C 180,E1 -10275.595,E2 -10275.595} C_VEL
LIN {X 0,Y 418.227,Z 458.867,A -85,B 0,C 180,E1 -10278.618,E2 -10278.618} C_VEL
LIN {X 0,Y 418.218,Z 458.883,A -85,B 0,C 180,E1 -10281.695,E2 -10281.695} C_VEL
LIN {X 0,Y 418.234,Z 458.882,A -85,B 0,C 180,E1 -10284.851,E2 -10284.851} C_VEL
LIN {X 0,Y 418.195,Z 458.879,A -85,B 0,C 180,E1 -10288.068,E2 -10288.068} C_VEL
LIN {X 0,Y 418.226,Z 458.886,A -85,B 0,C 180,E1 -10291.018,E2 -10291.018} C_VEL
LIN {X 0,Y 418.22,Z 458.884,A -85,B 0,C 180,E1 -10293.677,E2 -10293.677} C_VEL
LIN {X 0,Y 418.22,Z 458.887,A -85,B 0,C 180,E1 -10297.224,E2 -10297.224} C_VEL
LIN {X 0,Y 418.193,Z 458.881,A -85,B 0,C 180,E1 -10300.866,E2 -10300.866} C_VEL
LIN {X 0,Y 418.189,Z 458.894,A -85,B 0,C 180,E1 -10303.727,E2 -10303.727} C_VEL
LIN {X 0,Y 418.183,Z 458.873,A -85,B 0,C 180,E1 -10306.446,E2 -10306.446} C_VEL
LIN {X 0,Y 418.191,Z 458.873,A -85,B 0,C 180,E1 -10309.132,E2 -10309.132} C_VEL
LIN {X 0,Y 418.217,Z 458.887,A -85,B 0,C 180,E1 -10312.774,E2 -10312.774} C_VEL
LIN {X 0,Y 418.216,Z 458.876,A -85,B 0,C 180,E1 -10316.32,E2 -10316.32} C_VEL
LIN {X 0,Y 418.223,Z 458.882,A -85,B 0,C 180,E1 -10319.727,E2 -10319.727} C_VEL
LIN {X 0,Y 418.194,Z 458.892,A -85,B 0,C 180,E1 -10323.016,E2 -10323.016} C_VEL
LIN {X 0,Y 418.243,Z 458.89,A -85,B 0,C 180,E1 -10326.216,E2 -10326.216} C_VEL
LIN {X 0,Y 418.233,Z 458.889,A -85,B 0,C 180,E1 -10329.336,E2 -10329.336} C_VEL
LIN {X 0,Y 418.239,Z 458.889,A -85,B 0,C 180,E1 -10332.394,E2 -10332.394} C_VEL
LIN {X 0,Y 418.262,Z 458.887,A -85,B 0,C 180,E1 -10335.402,E2 -10335.402} C_VEL
LIN {X 0,Y 418.287,Z 458.884,A -85,B 0,C 180,E1 -10338.368,E2 -10338.368} C_VEL
LIN {X 0,Y 418.43,Z 458.866,A -85,B 0,C 180,E1 -10342.278,E2 -10342.278} C_VEL
LIN {X 0,Y 418.453,Z 458.863,A -85,B 0,C 180,E1 -10344.216,E2 -10344.216} C_VEL
LIN {X 0,Y 418.516,Z 458.855,A -85,B 0,C 180,E1 -10348.075,E2 -10348.075} C_VEL
LIN {X 0,Y 418.389,Z 458.87,A -85,B 0,C 180,E1 -10350.962,E2 -10350.962} C_VEL
LIN {X 0,Y 418.452,Z 458.862,A -85,B 0,C 180,E1 -10352.888,E2 -10352.888} C_VEL
LIN {X 0,Y 418.453,Z 458.863,A -85,B 0,C 180,E1 -10355.784,E2 -10355.784} C_VEL
LIN {X 0,Y 418.352,Z 458.875,A -85,B 0,C 180,E1 -10358.696,E2 -10358.696} C_VEL
LIN {X 0,Y 418.337,Z 458.877,A -85,B 0,C 180,E1 -10362.615,E2 -10362.615} C_VEL
LIN {X 0,Y 418.3,Z 458.881,A -85,B 0,C 180,E1 -10363.302,E2 -10363.302} C_VEL
LIN {X 0,Y 417.585,Z 458.972,A -85,B 0,C 180,E1 -10364.105,E2 -10364.105} C_VEL
LIN {X 0,Y 414.688,Z 459.331,A -85,B 0,C 180,E1 -10365.41,E2 -10365.41} C_VEL
LIN {X 0,Y 412.276,Z 459.632,A -85,B 0,C 180,E1 -10366.464,E2 -10366.464} C_VEL
LIN {X 0,Y 411.263,Z 459.758,A -85,B 0,C 180,E1 -10367.279,E2 -10367.279} C_VEL
LIN {X 0,Y 411.191,Z 459.766,A -85,B 0,C 180,E1 -10367.555,E2 -10367.555} C_VEL
LIN {X 0,Y 411.18,Z 459.767,A -85,B 0,C 180,E1 -10371.035,E2 -10371.035} C_VEL
LIN {X 0,Y 411.176,Z 459.769,A -85,B 0,C 180,E1 -10374.218,E2 -10374.218} C_VEL
LIN {X 0,Y 411.131,Z 459.774,A -85,B 0,C 180,E1 -10377.487,E2 -10377.487} C_VEL
LIN {X 0,Y 411.18,Z 459.753,A -85,B 0,C 180,E1 -10379.714,E2 -10379.714} C_VEL
LIN {X 0,Y 411.189,Z 459.76,A -85,B 0,C 180,E1 -10383.157,E2 -10383.157} C_VEL
LIN {X 0,Y 411.173,Z 459.765,A -85,B 0,C 180,E1 -10386.552,E2 -10386.552} C_VEL
LIN {X 0,Y 411.148,Z 459.761,A -85,B 0,C 180,E1 -10389.72,E2 -10389.72} C_VEL
LIN {X 0,Y 411.147,Z 459.746,A -85,B 0,C 180,E1 -10393.136,E2 -10393.136} C_VEL
LIN {X 0,Y 411.15,Z 459.77,A -85,B 0,C 180,E1 -10395.883,E2 -10395.883} C_VEL
LIN {X 0,Y 411.133,Z 459.761,A -85,B 0,C 180,E1 -10398.776,E2 -10398.776} C_VEL
LIN {X 0,Y 411.169,Z 459.772,A -85,B 0,C 180,E1 -10402.026,E2 -10402.026} C_VEL
LIN {X 0,Y 411.189,Z 459.752,A -85,B 0,C 180,E1 -10405.125,E2 -10405.125} C_VEL
LIN {X 0,Y 411.151,Z 459.772,A -85,B 0,C 180,E1 -10408.004,E2 -10408.004} C_VEL
LIN {X 0,Y 411.161,Z 459.762,A -85,B 0,C 180,E1 -10411.408,E2 -10411.408} C_VEL
LIN {X 0,Y 411.178,Z 459.761,A -85,B 0,C 180,E1 -10414.943,E2 -10414.943} C_VEL
LIN {X 0,Y 411.191,Z 459.763,A -85,B 0,C 180,E1 -10417.915,E2 -10417.915} C_VEL
LIN {X 0,Y 411.173,Z 459.744,A -85,B 0,C 180,E1 -10421.051,E2 -10421.051} C_VEL
LIN {X 0,Y 411.199,Z 459.766,A -85,B 0,C 180,E1 -10424.131,E2 -10424.131} C_VEL
LIN {X 0,Y 411.295,Z 459.746,A -85,B 0,C 180,E1 -10427.167,E2 -10427.167} C_VEL
LIN {X 0,Y 411.266,Z 459.735,A -85,B 0,C 180,E1 -10430.162,E2 -10430.162} C_VEL
LIN {X 0,Y 411.384,Z 459.735,A -85,B 0,C 180,E1 -10433.133,E2 -10433.133} C_VEL
LIN {X 0,Y 411.278,Z 459.751,A -85,B 0,C 180,E1 -10435.1,E2 -10435.1} C_VEL
LIN {X 0,Y 411.495,Z 459.71,A -85,B 0,C 180,E1 -10438.044,E2 -10438.044} C_VEL
LIN {X 0,Y 411.371,Z 459.726,A -85,B 0,C 180,E1 -10440.98,E2 -10440.98} C_VEL
LIN {X 0,Y 411.421,Z 459.731,A -85,B 0,C 180,E1 -10442.939,E2 -10442.939} C_VEL
LIN {X 0,Y 411.386,Z 459.731,A -85,B 0,C 180,E1 -10446.87,E2 -10446.87} C_VEL
LIN {X 0,Y 411.27,Z 459.733,A -85,B 0,C 180,E1 -10449.841,E2 -10449.841} C_VEL
LIN {X 0,Y 411.297,Z 459.746,A -85,B 0,C 180,E1 -10453.101,E2 -10453.101} C_VEL
LIN {X 0,Y 411.203,Z 459.749,A -85,B 0,C 180,E1 -10456.892,E2 -10456.892} C_VEL
LIN {X 0,Y 411.201,Z 459.751,A -85,B 0,C 180,E1 -10459.99,E2 -10459.99} C_VEL
LIN {X 0,Y 411.186,Z 459.762,A -85,B 0,C 180,E1 -10463.15,E2 -10463.15} C_VEL
LIN {X 0,Y 411.17,Z 459.749,A -85,B 0,C 180,E1 -10466.387,E2 -10466.387} C_VEL
LIN {X 0,Y 411.195,Z 459.764,A -85,B 0,C 180,E1 -10469.714,E2 -10469.714} C_VEL
LIN {X 0,Y 411.205,Z 459.753,A -85,B 0,C 180,E1 -10473.157,E2 -10473.157} C_VEL
LIN {X 0,Y 411.188,Z 459.764,A -85,B 0,C 180,E1 -10476.553,E2 -10476.553} C_VEL
LIN {X 0,Y 411.163,Z 459.762,A -85,B 0,C 180,E1 -10479.72,E2 -10479.72} C_VEL
LIN {X 0,Y 411.162,Z 459.766,A -85,B 0,C 180,E1 -10483.136,E2 -10483.136} C_VEL
LIN {X 0,Y 411.158,Z 459.773,A -85,B 0,C 180,E1 -10485.884,E2 -10485.884} C_VEL
LIN {X 0,Y 411.145,Z 459.753,A -85,B 0,C 180,E1 -10488.776,E2 -10488.776} C_VEL
LIN {X 0,Y 411.18,Z 459.767,A -85,B 0,C 180,E1 -10492.025,E2 -10492.025} C_VEL
LIN {X 0,Y 411.201,Z 459.762,A -85,B 0,C 180,E1 -10495.125,E2 -10495.125} C_VEL
LIN {X 0,Y 411.157,Z 459.768,A -85,B 0,C 180,E1 -10498.002,E2 -10498.002} C_VEL
LIN {X 0,Y 411.237,Z 459.927,A -85,B 0,C 180,E1 -10500.516,E2 -10500.516} C_VEL
LIN {X 0,Y 413.158,Z 470.054,A -85,B 0,C 180,E1 -10503.479,E2 -10503.479} C_VEL
LIN {X 0,Y 413.783,Z 475.268,A -85,B 0,C 180,E1 -10504.874,E2 -10504.874} C_VEL
LIN {X 0,Y 412.675,Z 489.764,A -85,B 0,C 180,E1 -10508.522,E2 -10508.522} C_VEL
LIN {X 0,Y 412.196,Z 497.652,A -85,B 0,C 180,E1 -10510.549,E2 -10510.549} C_VEL
LIN {X 0,Y 412.743,Z 501.113,A -85,B 0,C 180,E1 -10510.693,E2 -10510.693} C_VEL
LIN {X 0,Y 416.991,Z 525.194,A -85,B 0,C 180,E1 -10511.324,E2 -10511.324} C_VEL
LIN {X 0,Y 416.131,Z 602.61,A -85,B 0,C 180,E1 -10512.683,E2 -10512.683} C_VEL
LIN {X 0,Y 415.783,Z 612.528,A -85,B 0,C 180,E1 -10512.953,E2 -10512.953} C_VEL
LIN {X 0,Y 415.349,Z 622.517,A -85,B 0,C 180,E1 -10513.346,E2 -10513.346} C_VEL
LIN {X 0,Y 414.858,Z 630.905,A -85,B 0,C 180,E1 -10513.769,E2 -10513.769} C_VEL
LIN {X 0,Y 414.155,Z 642.021,A -85,B 0,C 180,E1 -10514.498,E2 -10514.498} C_VEL
LIN {X 0,Y 413.539,Z 651.025,A -85,B 0,C 180,E1 -10515.231,E2 -10515.231} C_VEL
LIN {X 0,Y 412.954,Z 659.408,A -85,B 0,C 180,E1 -10516.051,E2 -10516.051} C_VEL
LIN {X 0,Y 412.442,Z 667.181,A -85,B 0,C 180,E1 -10516.951,E2 -10516.951} C_VEL
LIN {X 0,Y 411.674,Z 675.977,A -85,B 0,C 180,E1 -10518.179,E2 -10518.179} C_VEL
LIN {X 0,Y 411.164,Z 681.967,A -85,B 0,C 180,E1 -10519.163,E2 -10519.163} C_VEL
LIN {X 0,Y 410.758,Z 688.28,A -85,B 0,C 180,E1 -10520.397,E2 -10520.397} C_VEL
LIN {X 0,Y 410.433,Z 693.554,A -85,B 0,C 180,E1 -10521.631,E2 -10521.631} C_VEL
LIN {X 0,Y 410.172,Z 698.648,A -85,B 0,C 180,E1 -10523.111,E2 -10523.111} C_VEL
LIN {X 0,Y 410.021,Z 702.611,A -85,B 0,C 180,E1 -10524.591,E2 -10524.591} C_VEL
LIN {X 0,Y 409.933,Z 705.543,A -85,B 0,C 180,E1 -10526.068,E2 -10526.068} C_VEL
LIN {X 0,Y 409.927,Z 707.041,A -85,B 0,C 180,E1 -10527.052,E2 -10527.052} C_VEL
LIN {X 0,Y 409.937,Z 708.563,A -85,B 0,C 180,E1 -10529.018,E2 -10529.018} C_VEL
LIN {X 0,Y 409.928,Z 708.841,A -85,B 0,C 180,E1 -10530,E2 -10530} C_VEL
LIN {X 0,Y 409.968,Z 707.969,A -85,B 0,C 180,E1 -10531.965,E2 -10531.965} C_VEL
LIN {X 0,Y 409.927,Z 707.041,A -85,B 0,C 180,E1 -10532.948,E2 -10532.948} C_VEL
LIN {X 0,Y 410.022,Z 703.7,A -85,B 0,C 180,E1 -10534.916,E2 -10534.916} C_VEL
LIN {X 0,Y 410.046,Z 700.573,A -85,B 0,C 180,E1 -10536.224,E2 -10536.224} C_VEL
LIN {X 0,Y 410.209,Z 697.133,A -85,B 0,C 180,E1 -10537.383,E2 -10537.383} C_VEL
LIN {X 0,Y 410.546,Z 691.558,A -85,B 0,C 180,E1 -10538.863,E2 -10538.863} C_VEL
LIN {X 0,Y 410.933,Z 685.904,A -85,B 0,C 180,E1 -10540.096,E2 -10540.096} C_VEL
LIN {X 0,Y 411.398,Z 679.098,A -85,B 0,C 180,E1 -10541.33,E2 -10541.33} C_VEL
LIN {X 0,Y 412.103,Z 670.881,A -85,B 0,C 180,E1 -10542.558,E2 -10542.558} C_VEL
LIN {X 0,Y 412.689,Z 663.052,A -85,B 0,C 180,E1 -10543.542,E2 -10543.542} C_VEL
LIN {X 0,Y 413.273,Z 654.606,A -85,B 0,C 180,E1 -10544.435,E2 -10544.435} C_VEL
LIN {X 0,Y 413.942,Z 645.202,A -85,B 0,C 180,E1 -10545.258,E2 -10545.258} C_VEL
LIN {X 0,Y 414.538,Z 636.812,A -85,B 0,C 180,E1 -10545.865,E2 -10545.865} C_VEL
LIN {X 0,Y 415.152,Z 626.305,A -85,B 0,C 180,E1 -10546.472,E2 -10546.472} C_VEL
LIN {X 0,Y 415.649,Z 615.972,A -85,B 0,C 180,E1 -10546.926,E2 -10546.926} C_VEL
LIN {X 0,Y 416.006,Z 605.252,A -85,B 0,C 180,E1 -10547.259,E2 -10547.259} C_VEL
LIN {X 0,Y 416.442,Z 584.27,A -85,B 0,C 180,E1 -10547.652,E2 -10547.652} C_VEL
LIN {X 0,Y 416.938,Z 524.571,A -85,B 0,C 180,E1 -10548.69,E2 -10548.69} C_VEL
LIN {X 0,Y 412.185,Z 497.93,A -85,B 0,C 180,E1 -10549.419,E2 -10549.419} C_VEL
LIN {X 0,Y 412.214,Z 496.614,A -85,B 0,C 180,E1 -10549.677,E2 -10549.677} C_VEL
LIN {X 0,Y 413.157,Z 483.768,A -85,B 0,C 180,E1 -10553.031,E2 -10553.031} C_VEL
LIN {X 0,Y 413.778,Z 474.25,A -85,B 0,C 180,E1 -10555.459,E2 -10555.459} C_VEL
LIN {X 0,Y 412.491,Z 466.323,A -85,B 0,C 180,E1 -10557.627,E2 -10557.627} C_VEL
LIN {X 0,Y 411.231,Z 459.856,A -85,B 0,C 180,E1 -10559.541,E2 -10559.541} C_VEL
LIN {X 0,Y 411.208,Z 459.757,A -85,B 0,C 180,E1 -10563.155,E2 -10563.155} C_VEL
LIN {X 0,Y 411.19,Z 459.757,A -85,B 0,C 180,E1 -10566.551,E2 -10566.551} C_VEL
LIN {X 0,Y 411.165,Z 459.76,A -85,B 0,C 180,E1 -10569.718,E2 -10569.718} C_VEL
LIN {X 0,Y 411.156,Z 459.766,A -85,B 0,C 180,E1 -10573.135,E2 -10573.135} C_VEL
LIN {X 0,Y 411.164,Z 459.764,A -85,B 0,C 180,E1 -10575.881,E2 -10575.881} C_VEL
LIN {X 0,Y 411.156,Z 459.766,A -85,B 0,C 180,E1 -10579.491,E2 -10579.491} C_VEL
LIN {X 0,Y 411.178,Z 459.766,A -85,B 0,C 180,E1 -10582.023,E2 -10582.023} C_VEL
LIN {X 0,Y 411.201,Z 459.754,A -85,B 0,C 180,E1 -10585.123,E2 -10585.123} C_VEL
LIN {X 0,Y 411.164,Z 459.764,A -85,B 0,C 180,E1 -10588.001,E2 -10588.001} C_VEL
LIN {X 0,Y 411.172,Z 459.762,A -85,B 0,C 180,E1 -10591.405,E2 -10591.405} C_VEL
LIN {X 0,Y 411.187,Z 459.756,A -85,B 0,C 180,E1 -10594.94,E2 -10594.94} C_VEL
LIN {X 0,Y 411.196,Z 459.765,A -85,B 0,C 180,E1 -10597.912,E2 -10597.912} C_VEL
LIN {X 0,Y 411.175,Z 459.745,A -85,B 0,C 180,E1 -10601.048,E2 -10601.048} C_VEL
LIN {X 0,Y 411.193,Z 459.759,A -85,B 0,C 180,E1 -10604.128,E2 -10604.128} C_VEL
LIN {X 0,Y 411.292,Z 459.746,A -85,B 0,C 180,E1 -10607.164,E2 -10607.164} C_VEL
LIN {X 0,Y 411.27,Z 459.733,A -85,B 0,C 180,E1 -10610.159,E2 -10610.159} C_VEL
LIN {X 0,Y 411.386,Z 459.731,A -85,B 0,C 180,E1 -10613.13,E2 -10613.13} C_VEL
LIN {X 0,Y 411.279,Z 459.751,A -85,B 0,C 180,E1 -10615.097,E2 -10615.097} C_VEL
LIN {X 0,Y 411.496,Z 459.719,A -85,B 0,C 180,E1 -10618.041,E2 -10618.041} C_VEL
LIN {X 0,Y 411.371,Z 459.72,A -85,B 0,C 180,E1 -10620.977,E2 -10620.977} C_VEL
LIN {X 0,Y 411.42,Z 459.728,A -85,B 0,C 180,E1 -10622.936,E2 -10622.936} C_VEL
LIN {X 0,Y 411.384,Z 459.735,A -85,B 0,C 180,E1 -10626.867,E2 -10626.867} C_VEL
LIN {X 0,Y 411.266,Z 459.735,A -85,B 0,C 180,E1 -10629.838,E2 -10629.838} C_VEL
LIN {X 0,Y 411.298,Z 459.745,A -85,B 0,C 180,E1 -10633.102,E2 -10633.102} C_VEL
LIN {X 0,Y 411.199,Z 459.756,A -85,B 0,C 180,E1 -10636.889,E2 -10636.889} C_VEL
LIN {X 0,Y 411.195,Z 459.746,A -85,B 0,C 180,E1 -10639.987,E2 -10639.987} C_VEL
LIN {X 0,Y 411.179,Z 459.763,A -85,B 0,C 180,E1 -10643.147,E2 -10643.147} C_VEL
LIN {X 0,Y 411.16,Z 459.755,A -85,B 0,C 180,E1 -10646.384,E2 -10646.384} C_VEL
LIN {X 0,Y 411.184,Z 459.761,A -85,B 0,C 180,E1 -10649.712,E2 -10649.712} C_VEL
LIN {X 0,Y 411.193,Z 459.758,A -85,B 0,C 180,E1 -10653.155,E2 -10653.155} C_VEL
LIN {X 0,Y 411.176,Z 459.766,A -85,B 0,C 180,E1 -10656.55,E2 -10656.55} C_VEL
LIN {X 0,Y 411.155,Z 459.766,A -85,B 0,C 180,E1 -10659.719,E2 -10659.719} C_VEL
LIN {X 0,Y 411.149,Z 459.768,A -85,B 0,C 180,E1 -10663.134,E2 -10663.134} C_VEL
LIN {X 0,Y 411.148,Z 459.756,A -85,B 0,C 180,E1 -10665.881,E2 -10665.881} C_VEL
LIN {X 0,Y 411.129,Z 459.746,A -85,B 0,C 180,E1 -10668.774,E2 -10668.774} C_VEL
LIN {X 0,Y 411.163,Z 459.773,A -85,B 0,C 180,E1 -10672.023,E2 -10672.023} C_VEL
LIN {X 0,Y 411.186,Z 459.744,A -85,B 0,C 180,E1 -10675.123,E2 -10675.123} C_VEL
LIN {X 0,Y 411.147,Z 459.773,A -85,B 0,C 180,E1 -10678.002,E2 -10678.002} C_VEL
LIN {X 0,Y 411.156,Z 459.758,A -85,B 0,C 180,E1 -10681.406,E2 -10681.406} C_VEL
LIN {X 0,Y 411.173,Z 459.767,A -85,B 0,C 180,E1 -10684.94,E2 -10684.94} C_VEL
LIN {X 0,Y 411.187,Z 459.769,A -85,B 0,C 180,E1 -10687.913,E2 -10687.913} C_VEL
LIN {X 0,Y 411.199,Z 459.765,A -85,B 0,C 180,E1 -10691.051,E2 -10691.051} C_VEL
LIN {X 0,Y 411.194,Z 459.767,A -85,B 0,C 180,E1 -10694.13,E2 -10694.13} C_VEL
LIN {X 0,Y 411.286,Z 459.754,A -85,B 0,C 180,E1 -10697.165,E2 -10697.165} C_VEL
LIN {X 0,Y 411.262,Z 459.759,A -85,B 0,C 180,E1 -10700.161,E2 -10700.161} C_VEL
LIN {X 0,Y 411.374,Z 459.745,A -85,B 0,C 180,E1 -10703.132,E2 -10703.132} C_VEL
LIN {X 0,Y 411.269,Z 459.758,A -85,B 0,C 180,E1 -10705.099,E2 -10705.099} C_VEL
LIN {X 0,Y 411.485,Z 459.731,A -85,B 0,C 180,E1 -10708.042,E2 -10708.042} C_VEL
LIN {X 0,Y 411.36,Z 459.746,A -85,B 0,C 180,E1 -10710.979,E2 -10710.979} C_VEL
LIN {X 0,Y 411.411,Z 459.74,A -85,B 0,C 180,E1 -10712.938,E2 -10712.938} C_VEL
LIN {X 0,Y 411.374,Z 459.745,A -85,B 0,C 180,E1 -10716.868,E2 -10716.868} C_VEL
LIN {X 0,Y 411.262,Z 459.759,A -85,B 0,C 180,E1 -10719.839,E2 -10719.839} C_VEL
LIN {X 0,Y 411.266,Z 459.757,A -85,B 0,C 180,E1 -10723.286,E2 -10723.286} C_VEL
LIN {X 0,Y 411.193,Z 459.766,A -85,B 0,C 180,E1 -10726.891,E2 -10726.891} C_VEL
LIN {X 0,Y 411.191,Z 459.766,A -85,B 0,C 180,E1 -10727.555,E2 -10727.555} C_VEL
LIN {X 0,Y 410.545,Z 459.849,A -85,B 0,C 180,E1 -10728.373,E2 -10728.373} C_VEL
LIN {X 0,Y 407.673,Z 460.207,A -85,B 0,C 180,E1 -10729.702,E2 -10729.702} C_VEL
LIN {X 0,Y 405.232,Z 460.509,A -85,B 0,C 180,E1 -10730.776,E2 -10730.776} C_VEL
LIN {X 0,Y 404.195,Z 460.639,A -85,B 0,C 180,E1 -10731.606,E2 -10731.606} C_VEL
LIN {X 0,Y 404.117,Z 460.646,A -85,B 0,C 180,E1 -10731.887,E2 -10731.887} C_VEL
LIN {X 0,Y 404.138,Z 460.645,A -85,B 0,C 180,E1 -10735.278,E2 -10735.278} C_VEL
LIN {X 0,Y 404.134,Z 460.629,A -85,B 0,C 180,E1 -10739.138,E2 -10739.138} C_VEL
LIN {X 0,Y 404.124,Z 460.641,A -85,B 0,C 180,E1 -10742.623,E2 -10742.623} C_VEL
LIN {X 0,Y 404.128,Z 460.624,A -85,B 0,C 180,E1 -10745.183,E2 -10745.183} C_VEL
LIN {X 0,Y 404.113,Z 460.644,A -85,B 0,C 180,E1 -10748.761,E2 -10748.761} C_VEL
LIN {X 0,Y 404.085,Z 460.618,A -85,B 0,C 180,E1 -10751.597,E2 -10751.597} C_VEL
LIN {X 0,Y 404.128,Z 460.638,A -85,B 0,C 180,E1 -10754.523,E2 -10754.523} C_VEL
LIN {X 0,Y 404.108,Z 460.646,A -85,B 0,C 180,E1 -10757.295,E2 -10757.295} C_VEL
LIN {X 0,Y 404.12,Z 460.638,A -85,B 0,C 180,E1 -10759.952,E2 -10759.952} C_VEL
LIN {X 0,Y 404.118,Z 460.644,A -85,B 0,C 180,E1 -10763.128,E2 -10763.128} C_VEL
LIN {X 0,Y 404.126,Z 460.636,A -85,B 0,C 180,E1 -10766.188,E2 -10766.188} C_VEL
LIN {X 0,Y 404.131,Z 460.647,A -85,B 0,C 180,E1 -10769.716,E2 -10769.716} C_VEL
LIN {X 0,Y 404.092,Z 460.631,A -85,B 0,C 180,E1 -10773.118,E2 -10773.118} C_VEL
LIN {X 0,Y 404.14,Z 460.642,A -85,B 0,C 180,E1 -10776.426,E2 -10776.426} C_VEL
LIN {X 0,Y 404.141,Z 460.625,A -85,B 0,C 180,E1 -10779.892,E2 -10779.892} C_VEL
LIN {X 0,Y 404.147,Z 460.634,A -85,B 0,C 180,E1 -10783.023,E2 -10783.023} C_VEL
LIN {X 0,Y 404.276,Z 460.62,A -85,B 0,C 180,E1 -10786.94,E2 -10786.94} C_VEL
LIN {X 0,Y 404.234,Z 460.609,A -85,B 0,C 180,E1 -10789.989,E2 -10789.989} C_VEL
LIN {X 0,Y 404.334,Z 460.613,A -85,B 0,C 180,E1 -10793.013,E2 -10793.013} C_VEL
LIN {X 0,Y 404.249,Z 460.627,A -85,B 0,C 180,E1 -10795.015,E2 -10795.015} C_VEL
LIN {X 0,Y 404.464,Z 460.586,A -85,B 0,C 180,E1 -10798.01,E2 -10798.01} C_VEL
LIN {X 0,Y 404.465,Z 460.595,A -85,B 0,C 180,E1 -10801.993,E2 -10801.993} C_VEL
LIN {X 0,Y 404.362,Z 460.613,A -85,B 0,C 180,E1 -10805.987,E2 -10805.987} C_VEL
LIN {X 0,Y 404.251,Z 460.604,A -85,B 0,C 180,E1 -10809.003,E2 -10809.003} C_VEL
LIN {X 0,Y 404.241,Z 460.625,A -85,B 0,C 180,E1 -10812.043,E2 -10812.043} C_VEL
LIN {X 0,Y 404.154,Z 460.636,A -85,B 0,C 180,E1 -10815.121,E2 -10815.121} C_VEL
LIN {X 0,Y 404.124,Z 460.623,A -85,B 0,C 180,E1 -10818.243,E2 -10818.243} C_VEL
LIN {X 0,Y 404.124,Z 460.639,A -85,B 0,C 180,E1 -10821.422,E2 -10821.422} C_VEL
LIN {X 0,Y 404.134,Z 460.634,A -85,B 0,C 180,E1 -10824.67,E2 -10824.67} C_VEL
LIN {X 0,Y 404.103,Z 460.637,A -85,B 0,C 180,E1 -10828.008,E2 -10828.008} C_VEL
LIN {X 0,Y 404.142,Z 460.643,A -85,B 0,C 180,E1 -10830.287,E2 -10830.287} C_VEL
LIN {X 0,Y 404.138,Z 460.631,A -85,B 0,C 180,E1 -10833.814,E2 -10833.814} C_VEL
LIN {X 0,Y 404.13,Z 460.642,A -85,B 0,C 180,E1 -10836.875,E2 -10836.875} C_VEL
LIN {X 0,Y 404.118,Z 460.64,A -85,B 0,C 180,E1 -10840.076,E2 -10840.076} C_VEL
LIN {X 0,Y 404.142,Z 460.64,A -85,B 0,C 180,E1 -10843.083,E2 -10843.083} C_VEL
LIN {X 0,Y 404.116,Z 460.65,A -85,B 0,C 180,E1 -10845.922,E2 -10845.922} C_VEL
LIN {X 0,Y 404.099,Z 460.63,A -85,B 0,C 180,E1 -10848.633,E2 -10848.633} C_VEL
LIN {X 0,Y 404.136,Z 460.644,A -85,B 0,C 180,E1 -10851.497,E2 -10851.497} C_VEL
LIN {X 0,Y 404.173,Z 460.637,A -85,B 0,C 180,E1 -10854.983,E2 -10854.983} C_VEL
LIN {X 0,Y 404.135,Z 460.648,A -85,B 0,C 180,E1 -10858.445,E2 -10858.445} C_VEL
LIN {X 0,Y 404.225,Z 460.824,A -85,B 0,C 180,E1 -10860.249,E2 -10860.249} C_VEL
LIN {X 0,Y 406.151,Z 470.911,A -85,B 0,C 180,E1 -10863.263,E2 -10863.263} C_VEL
LIN {X 0,Y 406.818,Z 476.128,A -85,B 0,C 180,E1 -10864.687,E2 -10864.687} C_VEL
LIN {X 0,Y 405.826,Z 489.592,A -85,B 0,C 180,E1 -10868.141,E2 -10868.141} C_VEL
LIN {X 0,Y 405.257,Z 497.453,A -85,B 0,C 180,E1 -10870.202,E2 -10870.202} C_VEL
LIN {X 0,Y 405.823,Z 500.921,A -85,B 0,C 180,E1 -10870.35,E2 -10870.35} C_VEL
LIN {X 0,Y 410.269,Z 525.915,A -85,B 0,C 180,E1 -10871.023,E2 -10871.023} C_VEL
LIN {X 0,Y 409.367,Z 602.414,A -85,B 0,C 180,E1 -10872.387,E2 -10872.387} C_VEL
LIN {X 0,Y 409.006,Z 612.332,A -85,B 0,C 180,E1 -10872.662,E2 -10872.662} C_VEL
LIN {X 0,Y 408.562,Z 622.321,A -85,B 0,C 180,E1 -10873.061,E2 -10873.061} C_VEL
LIN {X 0,Y 408.026,Z 630.708,A -85,B 0,C 180,E1 -10873.489,E2 -10873.489} C_VEL
LIN {X 0,Y 407.326,Z 641.825,A -85,B 0,C 180,E1 -10874.232,E2 -10874.232} C_VEL
LIN {X 0,Y 406.644,Z 650.828,A -85,B 0,C 180,E1 -10874.975,E2 -10874.975} C_VEL
LIN {X 0,Y 406.063,Z 658.725,A -85,B 0,C 180,E1 -10875.753,E2 -10875.753} C_VEL
LIN {X 0,Y 405.484,Z 666.984,A -85,B 0,C 180,E1 -10876.723,E2 -10876.723} C_VEL
LIN {X 0,Y 404.696,Z 675.78,A -85,B 0,C 180,E1 -10877.972,E2 -10877.972} C_VEL
LIN {X 0,Y 404.159,Z 681.77,A -85,B 0,C 180,E1 -10878.973,E2 -10878.973} C_VEL
LIN {X 0,Y 403.718,Z 688.083,A -85,B 0,C 180,E1 -10880.228,E2 -10880.228} C_VEL
LIN {X 0,Y 403.372,Z 693.357,A -85,B 0,C 180,E1 -10881.483,E2 -10881.483} C_VEL
LIN {X 0,Y 403.086,Z 698.451,A -85,B 0,C 180,E1 -10882.99,E2 -10882.99} C_VEL
LIN {X 0,Y 402.918,Z 702.414,A -85,B 0,C 180,E1 -10884.495,E2 -10884.495} C_VEL
LIN {X 0,Y 402.854,Z 705.346,A -85,B 0,C 180,E1 -10885.999,E2 -10885.999} C_VEL
LIN {X 0,Y 402.825,Z 706.845,A -85,B 0,C 180,E1 -10887,E2 -10887} C_VEL
LIN {X 0,Y 402.864,Z 708.367,A -85,B 0,C 180,E1 -10889,E2 -10889} C_VEL
LIN {X 0,Y 402.853,Z 708.645,A -85,B 0,C 180,E1 -10890,E2 -10890} C_VEL
LIN {X 0,Y 402.866,Z 707.773,A -85,B 0,C 180,E1 -10891.999,E2 -10891.999} C_VEL
LIN {X 0,Y 402.826,Z 706.845,A -85,B 0,C 180,E1 -10893,E2 -10893} C_VEL
LIN {X 0,Y 402.934,Z 703.503,A -85,B 0,C 180,E1 -10895.003,E2 -10895.003} C_VEL
LIN {X 0,Y 403.008,Z 699.879,A -85,B 0,C 180,E1 -10896.508,E2 -10896.508} C_VEL
LIN {X 0,Y 403.261,Z 695.147,A -85,B 0,C 180,E1 -10898.014,E2 -10898.014} C_VEL
LIN {X 0,Y 403.64,Z 689.175,A -85,B 0,C 180,E1 -10899.521,E2 -10899.521} C_VEL
LIN {X 0,Y 404.056,Z 683.082,A -85,B 0,C 180,E1 -10900.777,E2 -10900.777} C_VEL
LIN {X 0,Y 404.562,Z 677.341,A -85,B 0,C 180,E1 -10901.778,E2 -10901.778} C_VEL
LIN {X 0,Y 405.152,Z 670.684,A -85,B 0,C 180,E1 -10902.778,E2 -10902.778} C_VEL
LIN {X 0,Y 405.775,Z 662.855,A -85,B 0,C 180,E1 -10903.777,E2 -10903.777} C_VEL
LIN {X 0,Y 406.411,Z 653.717,A -85,B 0,C 180,E1 -10904.752,E2 -10904.752} C_VEL
LIN {X 0,Y 407.088,Z 645.005,A -85,B 0,C 180,E1 -10905.521,E2 -10905.521} C_VEL
LIN {X 0,Y 407.701,Z 636.615,A -85,B 0,C 180,E1 -10906.139,E2 -10906.139} C_VEL
LIN {X 0,Y 408.347,Z 626.108,A -85,B 0,C 180,E1 -10906.755,E2 -10906.755} C_VEL
LIN {X 0,Y 408.87,Z 615.776,A -85,B 0,C 180,E1 -10907.216,E2 -10907.216} C_VEL
LIN {X 0,Y 409.242,Z 605.056,A -85,B 0,C 180,E1 -10907.554,E2 -10907.554} C_VEL
LIN {X 0,Y 409.672,Z 582.283,A -85,B 0,C 180,E1 -10907.986,E2 -10907.986} C_VEL
LIN {X 0,Y 410.256,Z 525.715,A -85,B 0,C 180,E1 -10908.982,E2 -10908.982} C_VEL
LIN {X 0,Y 405.256,Z 498.065,A -85,B 0,C 180,E1 -10909.743,E2 -10909.743} C_VEL
LIN {X 0,Y 405.247,Z 496.91,A -85,B 0,C 180,E1 -10909.898,E2 -10909.898} C_VEL
LIN {X 0,Y 406.294,Z 483.241,A -85,B 0,C 180,E1 -10913.538,E2 -10913.538} C_VEL
LIN {X 0,Y 406.826,Z 475.354,A -85,B 0,C 180,E1 -10915.587,E2 -10915.587} C_VEL
LIN {X 0,Y 405.233,Z 466.003,A -85,B 0,C 180,E1 -10918.203,E2 -10918.203} C_VEL
LIN {X 0,Y 404.232,Z 460.738,A -85,B 0,C 180,E1 -10919.798,E2 -10919.798} C_VEL
LIN {X 0,Y 404.141,Z 460.642,A -85,B 0,C 180,E1 -10923.812,E2 -10923.812} C_VEL
LIN {X 0,Y 404.132,Z 460.639,A -85,B 0,C 180,E1 -10926.873,E2 -10926.873} C_VEL
LIN {X 0,Y 404.119,Z 460.631,A -85,B 0,C 180,E1 -10930.074,E2 -10930.074} C_VEL
LIN {X 0,Y 404.137,Z 460.64,A -85,B 0,C 180,E1 -10933.08,E2 -10933.08} C_VEL
LIN {X 0,Y 404.121,Z 460.641,A -85,B 0,C 180,E1 -10935.921,E2 -10935.921} C_VEL
LIN {X 0,Y 404.101,Z 460.645,A -85,B 0,C 180,E1 -10938.631,E2 -10938.631} C_VEL
LIN {X 0,Y 404.134,Z 460.638,A -85,B 0,C 180,E1 -10941.495,E2 -10941.495} C_VEL
LIN {X 0,Y 404.172,Z 460.629,A -85,B 0,C 180,E1 -10944.981,E2 -10944.981} C_VEL
LIN {X 0,Y 404.138,Z 460.644,A -85,B 0,C 180,E1 -10948.441,E2 -10948.441} C_VEL
LIN {X 0,Y 404.149,Z 460.637,A -85,B 0,C 180,E1 -10950.861,E2 -10950.861} C_VEL
LIN {X 0,Y 404.152,Z 460.633,A -85,B 0,C 180,E1 -10954.722,E2 -10954.722} C_VEL
LIN {X 0,Y 404.163,Z 460.638,A -85,B 0,C 180,E1 -10957.506,E2 -10957.506} C_VEL
LIN {X 0,Y 404.129,Z 460.623,A -85,B 0,C 180,E1 -10960.704,E2 -10960.704} C_VEL
LIN {X 0,Y 404.168,Z 460.629,A -85,B 0,C 180,E1 -10963.845,E2 -10963.845} C_VEL
LIN {X 0,Y 404.262,Z 460.622,A -85,B 0,C 180,E1 -10966.937,E2 -10966.937} C_VEL
LIN {X 0,Y 404.238,Z 460.609,A -85,B 0,C 180,E1 -10969.986,E2 -10969.986} C_VEL
LIN {X 0,Y 404.336,Z 460.609,A -85,B 0,C 180,E1 -10973.01,E2 -10973.01} C_VEL
LIN {X 0,Y 404.25,Z 460.626,A -85,B 0,C 180,E1 -10975.012,E2 -10975.012} C_VEL
LIN {X 0,Y 404.465,Z 460.595,A -85,B 0,C 180,E1 -10978.007,E2 -10978.007} C_VEL
LIN {X 0,Y 404.464,Z 460.586,A -85,B 0,C 180,E1 -10981.99,E2 -10981.99} C_VEL
LIN {X 0,Y 404.331,Z 460.615,A -85,B 0,C 180,E1 -10986.528,E2 -10986.528} C_VEL
LIN {X 0,Y 404.248,Z 460.611,A -85,B 0,C 180,E1 -10989,E2 -10989} C_VEL
LIN {X 0,Y 404.241,Z 460.619,A -85,B 0,C 180,E1 -10992.04,E2 -10992.04} C_VEL
LIN {X 0,Y 404.165,Z 460.637,A -85,B 0,C 180,E1 -10995.118,E2 -10995.118} C_VEL
LIN {X 0,Y 404.125,Z 460.626,A -85,B 0,C 180,E1 -10998.24,E2 -10998.24} C_VEL
LIN {X 0,Y 404.122,Z 460.636,A -85,B 0,C 180,E1 -11001.418,E2 -11001.418} C_VEL
LIN {X 0,Y 404.126,Z 460.641,A -85,B 0,C 180,E1 -11004.667,E2 -11004.667} C_VEL
LIN {X 0,Y 404.092,Z 460.634,A -85,B 0,C 180,E1 -11008.005,E2 -11008.005} C_VEL
LIN {X 0,Y 404.131,Z 460.647,A -85,B 0,C 180,E1 -11010.284,E2 -11010.284} C_VEL
LIN {X 0,Y 404.126,Z 460.636,A -85,B 0,C 180,E1 -11013.812,E2 -11013.812} C_VEL
LIN {X 0,Y 404.118,Z 460.644,A -85,B 0,C 180,E1 -11016.872,E2 -11016.872} C_VEL
LIN {X 0,Y 404.104,Z 460.639,A -85,B 0,C 180,E1 -11020.074,E2 -11020.074} C_VEL
LIN {X 0,Y 404.128,Z 460.642,A -85,B 0,C 180,E1 -11023.081,E2 -11023.081} C_VEL
LIN {X 0,Y 404.105,Z 460.632,A -85,B 0,C 180,E1 -11025.921,E2 -11025.921} C_VEL
LIN {X 0,Y 404.082,Z 460.621,A -85,B 0,C 180,E1 -11028.631,E2 -11028.631} C_VEL
LIN {X 0,Y 404.119,Z 460.644,A -85,B 0,C 180,E1 -11031.495,E2 -11031.495} C_VEL
LIN {X 0,Y 404.157,Z 460.62,A -85,B 0,C 180,E1 -11034.982,E2 -11034.982} C_VEL
LIN {X 0,Y 404.122,Z 460.646,A -85,B 0,C 180,E1 -11038.442,E2 -11038.442} C_VEL
LIN {X 0,Y 404.134,Z 460.629,A -85,B 0,C 180,E1 -11040.862,E2 -11040.862} C_VEL
LIN {X 0,Y 404.138,Z 460.645,A -85,B 0,C 180,E1 -11044.722,E2 -11044.722} C_VEL
LIN {X 0,Y 404.151,Z 460.644,A -85,B 0,C 180,E1 -11047.507,E2 -11047.507} C_VEL
LIN {X 0,Y 404.144,Z 460.645,A -85,B 0,C 180,E1 -11050.707,E2 -11050.707} C_VEL
LIN {X 0,Y 404.165,Z 460.643,A -85,B 0,C 180,E1 -11053.846,E2 -11053.846} C_VEL
LIN {X 0,Y 404.268,Z 460.629,A -85,B 0,C 180,E1 -11056.939,E2 -11056.939} C_VEL
LIN {X 0,Y 404.229,Z 460.635,A -85,B 0,C 180,E1 -11059.988,E2 -11059.988} C_VEL
LIN {X 0,Y 404.324,Z 460.623,A -85,B 0,C 180,E1 -11063.011,E2 -11063.011} C_VEL
LIN {X 0,Y 404.24,Z 460.633,A -85,B 0,C 180,E1 -11065.013,E2 -11065.013} C_VEL
LIN {X 0,Y 404.454,Z 460.607,A -85,B 0,C 180,E1 -11068.008,E2 -11068.008} C_VEL
LIN {X 0,Y 404.33,Z 460.622,A -85,B 0,C 180,E1 -11070.996,E2 -11070.996} C_VEL
LIN {X 0,Y 404.37,Z 460.617,A -85,B 0,C 180,E1 -11072.989,E2 -11072.989} C_VEL
LIN {X 0,Y 404.324,Z 460.623,A -85,B 0,C 180,E1 -11076.989,E2 -11076.989} C_VEL
LIN {X 0,Y 404.229,Z 460.635,A -85,B 0,C 180,E1 -11080.012,E2 -11080.012} C_VEL
LIN {X 0,Y 404.251,Z 460.631,A -85,B 0,C 180,E1 -11083.212,E2 -11083.212} C_VEL
LIN {X 0,Y 404.165,Z 460.642,A -85,B 0,C 180,E1 -11087.194,E2 -11087.194} C_VEL
LIN {X 0,Y 404.148,Z 460.645,A -85,B 0,C 180,E1 -11090.352,E2 -11090.352} C_VEL
LIN {X 0,Y 404.117,Z 460.646,A -85,B 0,C 180,E1 -11091.887,E2 -11091.887} C_VEL
LIN {X 0,Y 403.474,Z 460.728,A -85,B 0,C 180,E1 -11092.719,E2 -11092.719} C_VEL
LIN {X 0,Y 400.648,Z 461.085,A -85,B 0,C 180,E1 -11094.07,E2 -11094.07} C_VEL
LIN {X 0,Y 398.226,Z 461.389,A -85,B 0,C 180,E1 -11095.162,E2 -11095.162} C_VEL
LIN {X 0,Y 397.159,Z 461.518,A -85,B 0,C 180,E1 -11096.005,E2 -11096.005} C_VEL
LIN {X 0,Y 397.059,Z 461.528,A -85,B 0,C 180,E1 -11096.291,E2 -11096.291} C_VEL
LIN {X 0,Y 397.082,Z 461.509,A -85,B 0,C 180,E1 -11099.863,E2 -11099.863} C_VEL
LIN {X 0,Y 397.097,Z 461.511,A -85,B 0,C 180,E1 -11103.274,E2 -11103.274} C_VEL
LIN {X 0,Y 397.077,Z 461.52,A -85,B 0,C 180,E1 -11106.997,E2 -11106.997} C_VEL
LIN {X 0,Y 397.04,Z 461.508,A -85,B 0,C 180,E1 -11110.438,E2 -11110.438} C_VEL
LIN {X 0,Y 397.072,Z 461.501,A -85,B 0,C 180,E1 -11113.652,E2 -11113.652} C_VEL
LIN {X 0,Y 397.078,Z 461.522,A -85,B 0,C 180,E1 -11116.524,E2 -11116.524} C_VEL
LIN {X 0,Y 397.073,Z 461.522,A -85,B 0,C 180,E1 -11120.421,E2 -11120.421} C_VEL
LIN {X 0,Y 397.081,Z 461.52,A -85,B 0,C 180,E1 -11123.006,E2 -11123.006} C_VEL
LIN {X 0,Y 397.1,Z 461.514,A -85,B 0,C 180,E1 -11126.728,E2 -11126.728} C_VEL
LIN {X 0,Y 397.105,Z 461.514,A -85,B 0,C 180,E1 -11130.296,E2 -11130.296} C_VEL
LIN {X 0,Y 397.064,Z 461.511,A -85,B 0,C 180,E1 -11133.739,E2 -11133.739} C_VEL
LIN {X 0,Y 397.09,Z 461.519,A -85,B 0,C 180,E1 -11137.087,E2 -11137.087} C_VEL
LIN {X 0,Y 397.087,Z 461.499,A -85,B 0,C 180,E1 -11140.352,E2 -11140.352} C_VEL
LIN {X 0,Y 397.111,Z 461.513,A -85,B 0,C 180,E1 -11143.553,E2 -11143.553} C_VEL
LIN {X 0,Y 397.223,Z 461.499,A -85,B 0,C 180,E1 -11146.704,E2 -11146.704} C_VEL
LIN {X 0,Y 397.196,Z 461.485,A -85,B 0,C 180,E1 -11149.81,E2 -11149.81} C_VEL
LIN {X 0,Y 397.287,Z 461.491,A -85,B 0,C 180,E1 -11152.888,E2 -11152.888} C_VEL
LIN {X 0,Y 397.221,Z 461.502,A -85,B 0,C 180,E1 -11154.926,E2 -11154.926} C_VEL
LIN {X 0,Y 397.432,Z 461.462,A -85,B 0,C 180,E1 -11157.975,E2 -11157.975} C_VEL
LIN {X 0,Y 397.432,Z 461.471,A -85,B 0,C 180,E1 -11162.028,E2 -11162.028} C_VEL
LIN {X 0,Y 397.315,Z 461.489,A -85,B 0,C 180,E1 -11166.094,E2 -11166.094} C_VEL
LIN {X 0,Y 397.223,Z 461.479,A -85,B 0,C 180,E1 -11169.164,E2 -11169.164} C_VEL
LIN {X 0,Y 397.204,Z 461.505,A -85,B 0,C 180,E1 -11172.26,E2 -11172.26} C_VEL
LIN {X 0,Y 397.106,Z 461.515,A -85,B 0,C 180,E1 -11175.396,E2 -11175.396} C_VEL
LIN {X 0,Y 397.079,Z 461.5,A -85,B 0,C 180,E1 -11178.579,E2 -11178.579} C_VEL
LIN {X 0,Y 397.086,Z 461.52,A -85,B 0,C 180,E1 -11181.82,E2 -11181.82} C_VEL
LIN {X 0,Y 397.102,Z 461.51,A -85,B 0,C 180,E1 -11185.137,E2 -11185.137} C_VEL
LIN {X 0,Y 397.062,Z 461.52,A -85,B 0,C 180,E1 -11188.55,E2 -11188.55} C_VEL
LIN {X 0,Y 397.08,Z 461.52,A -85,B 0,C 180,E1 -11191.837,E2 -11191.837} C_VEL
LIN {X 0,Y 397.116,Z 461.508,A -85,B 0,C 180,E1 -11194.496,E2 -11194.496} C_VEL
LIN {X 0,Y 397.087,Z 461.517,A -85,B 0,C 180,E1 -11198.278,E2 -11198.278} C_VEL
LIN {X 0,Y 397.047,Z 461.522,A -85,B 0,C 180,E1 -11200.915,E2 -11200.915} C_VEL
LIN {X 0,Y 397.088,Z 461.519,A -85,B 0,C 180,E1 -11203.652,E2 -11203.652} C_VEL
LIN {X 0,Y 397.089,Z 461.52,A -85,B 0,C 180,E1 -11206.525,E2 -11206.525} C_VEL
LIN {X 0,Y 397.087,Z 461.514,A -85,B 0,C 180,E1 -11210.42,E2 -11210.42} C_VEL
LIN {X 0,Y 397.094,Z 461.516,A -85,B 0,C 180,E1 -11213.005,E2 -11213.005} C_VEL
LIN {X 0,Y 397.112,Z 461.513,A -85,B 0,C 180,E1 -11216.727,E2 -11216.727} C_VEL
LIN {X 0,Y 397.167,Z 461.667,A -85,B 0,C 180,E1 -11219.944,E2 -11219.944} C_VEL
LIN {X 0,Y 399.293,Z 472.815,A -85,B 0,C 180,E1 -11223.332,E2 -11223.332} C_VEL
LIN {X 0,Y 399.862,Z 476.987,A -85,B 0,C 180,E1 -11224.494,E2 -11224.494} C_VEL
LIN {X 0,Y 398.884,Z 489.418,A -85,B 0,C 180,E1 -11227.74,E2 -11227.74} C_VEL
LIN {X 0,Y 398.315,Z 497.272,A -85,B 0,C 180,E1 -11229.846,E2 -11229.846} C_VEL
LIN {X 0,Y 399.093,Z 501.709,A -85,B 0,C 180,E1 -11230.023,E2 -11230.023} C_VEL
LIN {X 0,Y 403.541,Z 526.713,A -85,B 0,C 180,E1 -11230.712,E2 -11230.712} C_VEL
LIN {X 0,Y 402.616,Z 602.218,A -85,B 0,C 180,E1 -11232.082,E2 -11232.082} C_VEL
LIN {X 0,Y 402.223,Z 612.135,A -85,B 0,C 180,E1 -11232.36,E2 -11232.36} C_VEL
LIN {X 0,Y 401.788,Z 622.125,A -85,B 0,C 180,E1 -11232.767,E2 -11232.767} C_VEL
LIN {X 0,Y 401.223,Z 630.512,A -85,B 0,C 180,E1 -11233.201,E2 -11233.201} C_VEL
LIN {X 0,Y 400.494,Z 641.629,A -85,B 0,C 180,E1 -11233.956,E2 -11233.956} C_VEL
LIN {X 0,Y 399.768,Z 650.631,A -85,B 0,C 180,E1 -11234.71,E2 -11234.71} C_VEL
LIN {X 0,Y 399.068,Z 659.463,A -85,B 0,C 180,E1 -11235.608,E2 -11235.608} C_VEL
LIN {X 0,Y 398.515,Z 666.836,A -85,B 0,C 180,E1 -11236.494,E2 -11236.494} C_VEL
LIN {X 0,Y 397.727,Z 675.583,A -85,B 0,C 180,E1 -11237.758,E2 -11237.758} C_VEL
LIN {X 0,Y 397.163,Z 681.573,A -85,B 0,C 180,E1 -11238.776,E2 -11238.776} C_VEL
LIN {X 0,Y 396.684,Z 687.885,A -85,B 0,C 180,E1 -11240.053,E2 -11240.053} C_VEL
LIN {X 0,Y 396.329,Z 693.16,A -85,B 0,C 180,E1 -11241.331,E2 -11241.331} C_VEL
LIN {X 0,Y 396.015,Z 698.254,A -85,B 0,C 180,E1 -11242.864,E2 -11242.864} C_VEL
LIN {X 0,Y 395.83,Z 701.79,A -85,B 0,C 180,E1 -11244.196,E2 -11244.196} C_VEL
LIN {X 0,Y 395.777,Z 705.15,A -85,B 0,C 180,E1 -11245.927,E2 -11245.927} C_VEL
LIN {X 0,Y 395.729,Z 706.648,A -85,B 0,C 180,E1 -11246.946,E2 -11246.946} C_VEL
LIN {X 0,Y 395.793,Z 708.172,A -85,B 0,C 180,E1 -11248.983,E2 -11248.983} C_VEL
LIN {X 0,Y 395.78,Z 708.45,A -85,B 0,C 180,E1 -11250,E2 -11250} C_VEL
LIN {X 0,Y 395.764,Z 707.576,A -85,B 0,C 180,E1 -11252.035,E2 -11252.035} C_VEL
LIN {X 0,Y 395.729,Z 706.648,A -85,B 0,C 180,E1 -11253.054,E2 -11253.054} C_VEL
LIN {X 0,Y 395.847,Z 703.307,A -85,B 0,C 180,E1 -11255.093,E2 -11255.093} C_VEL
LIN {X 0,Y 395.924,Z 699.682,A -85,B 0,C 180,E1 -11256.625,E2 -11256.625} C_VEL
LIN {X 0,Y 396.208,Z 694.95,A -85,B 0,C 180,E1 -11258.158,E2 -11258.158} C_VEL
LIN {X 0,Y 396.619,Z 688.979,A -85,B 0,C 180,E1 -11259.691,E2 -11259.691} C_VEL
LIN {X 0,Y 397.046,Z 682.885,A -85,B 0,C 180,E1 -11260.969,E2 -11260.969} C_VEL
LIN {X 0,Y 397.594,Z 677.144,A -85,B 0,C 180,E1 -11261.987,E2 -11261.987} C_VEL
LIN {X 0,Y 398.208,Z 670.488,A -85,B 0,C 180,E1 -11263.004,E2 -11263.004} C_VEL
LIN {X 0,Y 398.874,Z 662.661,A -85,B 0,C 180,E1 -11264.02,E2 -11264.02} C_VEL
LIN {X 0,Y 399.431,Z 654.965,A -85,B 0,C 180,E1 -11264.872,E2 -11264.872} C_VEL
LIN {X 0,Y 400.219,Z 644.808,A -85,B 0,C 180,E1 -11265.794,E2 -11265.794} C_VEL
LIN {X 0,Y 400.889,Z 636.419,A -85,B 0,C 180,E1 -11266.421,E2 -11266.421} C_VEL
LIN {X 0,Y 401.544,Z 625.912,A -85,B 0,C 180,E1 -11267.047,E2 -11267.047} C_VEL
LIN {X 0,Y 402.055,Z 615.579,A -85,B 0,C 180,E1 -11267.517,E2 -11267.517} C_VEL
LIN {X 0,Y 402.492,Z 604.86,A -85,B 0,C 180,E1 -11267.858,E2 -11267.858} C_VEL
LIN {X 0,Y 402.914,Z 582.086,A -85,B 0,C 180,E1 -11268.299,E2 -11268.299} C_VEL
LIN {X 0,Y 403.501,Z 526.367,A -85,B 0,C 180,E1 -11269.296,E2 -11269.296} C_VEL
LIN {X 0,Y 398.338,Z 497.756,A -85,B 0,C 180,E1 -11270.107,E2 -11270.107} C_VEL
LIN {X 0,Y 398.295,Z 496.715,A -85,B 0,C 180,E1 -11270.261,E2 -11270.261} C_VEL
LIN {X 0,Y 399.406,Z 483.423,A -85,B 0,C 180,E1 -11273.873,E2 -11273.873} C_VEL
LIN {X 0,Y 399.836,Z 476.214,A -85,B 0,C 180,E1 -11275.787,E2 -11275.787} C_VEL
LIN {X 0,Y 398.184,Z 466.86,A -85,B 0,C 180,E1 -11278.46,E2 -11278.46} C_VEL
LIN {X 0,Y 397.146,Z 461.62,A -85,B 0,C 180,E1 -11280.092,E2 -11280.092} C_VEL
LIN {X 0,Y 397.101,Z 461.518,A -85,B 0,C 180,E1 -11283.712,E2 -11283.712} C_VEL
LIN {X 0,Y 397.089,Z 461.517,A -85,B 0,C 180,E1 -11287.206,E2 -11287.206} C_VEL
LIN {X 0,Y 397.056,Z 461.507,A -85,B 0,C 180,E1 -11290.436,E2 -11290.436} C_VEL
LIN {X 0,Y 397.085,Z 461.521,A -85,B 0,C 180,E1 -11293.65,E2 -11293.65} C_VEL
LIN {X 0,Y 397.092,Z 461.52,A -85,B 0,C 180,E1 -11296.522,E2 -11296.522} C_VEL
LIN {X 0,Y 397.085,Z 461.515,A -85,B 0,C 180,E1 -11300.418,E2 -11300.418} C_VEL
LIN {X 0,Y 397.092,Z 461.519,A -85,B 0,C 180,E1 -11303.003,E2 -11303.003} C_VEL
LIN {X 0,Y 397.112,Z 461.508,A -85,B 0,C 180,E1 -11306.726,E2 -11306.726} C_VEL
LIN {X 0,Y 397.115,Z 461.517,A -85,B 0,C 180,E1 -11310.294,E2 -11310.294} C_VEL
LIN {X 0,Y 397.074,Z 461.504,A -85,B 0,C 180,E1 -11313.736,E2 -11313.736} C_VEL
LIN {X 0,Y 397.098,Z 461.516,A -85,B 0,C 180,E1 -11317.084,E2 -11317.084} C_VEL
LIN {X 0,Y 397.091,Z 461.503,A -85,B 0,C 180,E1 -11320.349,E2 -11320.349} C_VEL
LIN {X 0,Y 397.112,Z 461.505,A -85,B 0,C 180,E1 -11323.549,E2 -11323.549} C_VEL
LIN {X 0,Y 397.189,Z 461.504,A -85,B 0,C 180,E1 -11326.7,E2 -11326.7} C_VEL
LIN {X 0,Y 397.2,Z 461.487,A -85,B 0,C 180,E1 -11329.807,E2 -11329.807} C_VEL
LIN {X 0,Y 397.289,Z 461.487,A -85,B 0,C 180,E1 -11332.885,E2 -11332.885} C_VEL
LIN {X 0,Y 397.222,Z 461.502,A -85,B 0,C 180,E1 -11334.923,E2 -11334.923} C_VEL
LIN {X 0,Y 397.432,Z 461.471,A -85,B 0,C 180,E1 -11337.972,E2 -11337.972} C_VEL
LIN {X 0,Y 397.432,Z 461.462,A -85,B 0,C 180,E1 -11342.025,E2 -11342.025} C_VEL
LIN {X 0,Y 397.287,Z 461.493,A -85,B 0,C 180,E1 -11346.523,E2 -11346.523} C_VEL
LIN {X 0,Y 397.219,Z 461.486,A -85,B 0,C 180,E1 -11349.161,E2 -11349.161} C_VEL
LIN {X 0,Y 397.206,Z 461.498,A -85,B 0,C 180,E1 -11352.257,E2 -11352.257} C_VEL
LIN {X 0,Y 397.114,Z 461.517,A -85,B 0,C 180,E1 -11355.393,E2 -11355.393} C_VEL
LIN {X 0,Y 397.078,Z 461.5,A -85,B 0,C 180,E1 -11358.576,E2 -11358.576} C_VEL
LIN {X 0,Y 397.082,Z 461.516,A -85,B 0,C 180,E1 -11361.817,E2 -11361.817} C_VEL
LIN {X 0,Y 397.093,Z 461.516,A -85,B 0,C 180,E1 -11365.134,E2 -11365.134} C_VEL
LIN {X 0,Y 397.052,Z 461.517,A -85,B 0,C 180,E1 -11368.547,E2 -11368.547} C_VEL
LIN {X 0,Y 397.069,Z 461.527,A -85,B 0,C 180,E1 -11371.834,E2 -11371.834} C_VEL
LIN {X 0,Y 397.104,Z 461.506,A -85,B 0,C 180,E1 -11374.493,E2 -11374.493} C_VEL
LIN {X 0,Y 397.077,Z 461.524,A -85,B 0,C 180,E1 -11378.275,E2 -11378.275} C_VEL
LIN {X 0,Y 397.038,Z 461.522,A -85,B 0,C 180,E1 -11381.975,E2 -11381.975} C_VEL
LIN {X 0,Y 397.07,Z 461.517,A -85,B 0,C 180,E1 -11385.068,E2 -11385.068} C_VEL
LIN {X 0,Y 397.034,Z 461.494,A -85,B 0,C 180,E1 -11388.023,E2 -11388.023} C_VEL
LIN {X 0,Y 397.073,Z 461.521,A -85,B 0,C 180,E1 -11391.145,E2 -11391.145} C_VEL
LIN {X 0,Y 397.082,Z 461.503,A -85,B 0,C 180,E1 -11394.5,E2 -11394.5} C_VEL
LIN {X 0,Y 397.061,Z 461.526,A -85,B 0,C 180,E1 -11397.927,E2 -11397.927} C_VEL
LIN {X 0,Y 397.1,Z 461.505,A -85,B 0,C 180,E1 -11400.294,E2 -11400.294} C_VEL
LIN {X 0,Y 397.061,Z 461.528,A -85,B 0,C 180,E1 -11403.737,E2 -11403.737} C_VEL
LIN {X 0,Y 397.084,Z 461.523,A -85,B 0,C 180,E1 -11407.084,E2 -11407.084} C_VEL
LIN {X 0,Y 397.13,Z 461.519,A -85,B 0,C 180,E1 -11410.352,E2 -11410.352} C_VEL
LIN {X 0,Y 397.112,Z 461.521,A -85,B 0,C 180,E1 -11413.551,E2 -11413.551} C_VEL
LIN {X 0,Y 397.214,Z 461.509,A -85,B 0,C 180,E1 -11416.702,E2 -11416.702} C_VEL
LIN {X 0,Y 397.19,Z 461.513,A -85,B 0,C 180,E1 -11419.808,E2 -11419.808} C_VEL
LIN {X 0,Y 397.277,Z 461.502,A -85,B 0,C 180,E1 -11422.887,E2 -11422.887} C_VEL
LIN {X 0,Y 397.211,Z 461.509,A -85,B 0,C 180,E1 -11424.925,E2 -11424.925} C_VEL
LIN {X 0,Y 397.417,Z 461.805,A -85,B 0,C 180,E1 -11428.227,E2 -11428.227} C_VEL
LIN {X 0,Y 397.468,Z 462.072,A -85,B 0,C 180,E1 -11430,E2 -11430} C_VEL
LIN {X 0,Y 397.357,Z 461.612,A -85,B 0,C 180,E1 -11432.788,E2 -11432.788} C_VEL
LIN {X 0,Y 397.303,Z 461.497,A -85,B 0,C 180,E1 -11436.093,E2 -11436.093} C_VEL
LIN {X 0,Y 397.212,Z 461.508,A -85,B 0,C 180,E1 -11439.163,E2 -11439.163} C_VEL
LIN {X 0,Y 397.198,Z 461.51,A -85,B 0,C 180,E1 -11442.259,E2 -11442.259} C_VEL
LIN {X 0,Y 397.108,Z 461.521,A -85,B 0,C 180,E1 -11445.395,E2 -11445.395} C_VEL
LIN {X 0,Y 397.135,Z 461.518,A -85,B 0,C 180,E1 -11448.575,E2 -11448.575} C_VEL
LIN {X 0,Y 397.076,Z 461.526,A -85,B 0,C 180,E1 -11451.879,E2 -11451.879} C_VEL
LIN {X 0,Y 397.088,Z 461.522,A -85,B 0,C 180,E1 -11455.136,E2 -11455.136} C_VEL
LIN {X 0,Y 397.059,Z 461.528,A -85,B 0,C 180,E1 -11456.291,E2 -11456.291} C_VEL
LIN {X 0,Y 396.358,Z 461.615,A -85,B 0,C 180,E1 -11457.138,E2 -11457.138} C_VEL
LIN {X 0,Y 393.507,Z 461.957,A -85,B 0,C 180,E1 -11458.515,E2 -11458.515} C_VEL
LIN {X 0,Y 391.113,Z 462.254,A -85,B 0,C 180,E1 -11459.627,E2 -11459.627} C_VEL
LIN {X 0,Y 390.081,Z 462.388,A -85,B 0,C 180,E1 -11460.487,E2 -11460.487} C_VEL
LIN {X 0,Y 389.994,Z 462.397,A -85,B 0,C 180,E1 -11460.778,E2 -11460.778} C_VEL
LIN {X 0,Y 390.055,Z 462.376,A -85,B 0,C 180,E1 -11464.025,E2 -11464.025} C_VEL
LIN {X 0,Y 390.019,Z 462.404,A -85,B 0,C 180,E1 -11467.782,E2 -11467.782} C_VEL
LIN {X 0,Y 390,Z 462.38,A -85,B 0,C 180,E1 -11470.815,E2 -11470.815} C_VEL
LIN {X 0,Y 390.029,Z 462.381,A -85,B 0,C 180,E1 -11473.885,E2 -11473.885} C_VEL
LIN {X 0,Y 390.034,Z 462.398,A -85,B 0,C 180,E1 -11476.789,E2 -11476.789} C_VEL
LIN {X 0,Y 389.997,Z 462.393,A -85,B 0,C 180,E1 -11479.556,E2 -11479.556} C_VEL
LIN {X 0,Y 390.025,Z 462.401,A -85,B 0,C 180,E1 -11482.452,E2 -11482.452} C_VEL
LIN {X 0,Y 390.05,Z 462.387,A -85,B 0,C 180,E1 -11486.046,E2 -11486.046} C_VEL
